(*sensore di presenza alla base dell'ascensore*)
IF NOT (ReadyLoadForVerificationBlockHigh OR ReadyLoadForVerificationBlockLow) AND NOT RotaryMakerInPositionVerificationBlockLow  THEN
	IF LiftPosition<=8 AND ElementVerificationCharged OR (RotaryMakerInPositionVerification AND ElementRotaryCharged)  THEN
			ReadyLoadForVerification:=TRUE;  (*sensore di presenza alla base dell'ascensore*)
		ELSE ReadyLoadForVerification:=FALSE;
	END_IF;
END_IF;
(*caso RotaryMakerInPositionVerificationBlockLow*)
IF NOT (ReadyLoadForVerificationBlockHigh OR ReadyLoadForVerificationBlockLow) AND RotaryMakerInPositionVerificationBlockLow THEN
	IF LiftPosition<=8 AND ElementRotaryCharged AND RotaryPosition=180 THEN
			ReadyLoadForVerification:=TRUE;
	END_IF;
	IF  LiftPosition>8 OR ToExtendCylinderOfExtractionVsGuide THEN
			ReadyLoadForVerification:=FALSE;
	END_IF;
END_IF;

(*sensore di presenza alla base dell'ascensore guasto: *)
IF ReadyLoadForVerificationBlockHigh THEN
	ReadyLoadForVerification:=TRUE;
END_IF;
IF ReadyLoadForVerificationBlockLow THEN
	ReadyLoadForVerification:=FALSE;
END_IF;

(*visualizzazione ElementoMisura*)
IF CylinderUpToMeasureLoad (*.........AND NOT ElementOneTableCharged.........*) AND ElementVerificationCharged AND NOT CylinderUpToMeasureLoadBlockHigh THEN	(*Quando l'ascensore arriva in cima viene reso visibile l'elemento in questa posizione e invisibile quello in posizione di verifica*)
	ElementMeasureCharged:=TRUE;
	ElementMeasureRed:=ElementVerificationRed;
	ElementMeasureSilver:=ElementVerificationSilver;
	ElementMeasureBlack:=ElementVerificationBlack;
	ElementMeasureOverturned:=ElementVerificationOverturned;
	ElementMeasureShort:=ElementVerificationShort;
	ElementVerificationCharged:=FALSE;
END_IF;

(*cuscinetto d'aria*)
IF NOT AirCushionBlock THEN
	IF AirCushion THEN
			 AirCushionVis:=TRUE; (*visualizzazione cuscinetto*)
		ELSE IF NOT AirCushionBlockHigh THEN
				AirCushionVis:=FALSE;
			END_IF;
	END_IF;
END_IF;

(*Elemento cuscinetto d'aria*)
IF (AirCushionVis OR AirCushionBlock) AND (CylinderOfExtractionPosition=80)  THEN	(*Quando e' attiva l'aria dello scivolo e ho spinto il pezzo, viene reso visibile l'elemento in questa posizione e invisibile quello in posizione di misura*)
	ElementAirCharged:=TRUE;
	ElementAirRed:=ElementMeasureRed;
	ElementAirSilver:=ElementMeasureSilver;
	ElementAirBlack:=ElementMeasureBlack;
	ElementAirOverturned:=ElementMeasureOverturned;
	ElementMeasureCharged:=FALSE;
END_IF;

IF (AirCushionVis AND NOT AirCushionBlock) AND (CylinderOfExtractionPosition=80)  AND MovementElementAir<=20  THEN (*Quando l'aria  dello scivolo e' attiva e il pezzo è stato spinto, il pezzo va verso la tavola rotante*)
		MovementElementAir:=MovementElementAir+3;
	ELSE MovementElementAir:=0;
END_IF;

IF (MovementElementAir>=20)
THEN	MovementElementAir:=20;
		ElementAirVsRotaryTable:=TRUE;
		AirCushion:=FALSE;
		ElementAirCharged:=FALSE;
END_IF;

IF NOT Alligneed AND NOT ElementMeasureCharged
THEN	ElementAirRed:=FALSE;
		ElementAirSilver:=FALSE;
		ElementAirBlack:=FALSE;
		ElementMeasureRed:=FALSE;
		ElementMeasureSilver:=FALSE;
		ElementMeasureBlack:=FALSE;
END_IF;

(*---------------------------------------------------------*)
IF (Reset AND NOT MachineNOTOkForReset) OR Remove OR FaultDetected THEN  (*rimozione di tutti i pezzi presenti sulle macchine tramite pulsante o reset del sistema*)
	ElementOneCharged:=FALSE;
	ElementOneRed:=FALSE;
	ElementOneSilver:=FALSE;
	ElementOneBlack:=FALSE;
	ElementOneOverturned:=FALSE;
	ElementOneShort:=FALSE;
	ElementTwoCharged:=FALSE;
	ElementTwoRed:=FALSE;
	ElementTwoSilver:=FALSE;
	ElementTwoBlack:=FALSE;
	ElementTwoOverturned:=FALSE;
	ElementTwoShort:=FALSE;
	ElementThreeCharged:=FALSE;
	ElementThreeRed:=FALSE;
	ElementThreeSilver:=FALSE;
	ElementThreeBlack:=FALSE;
	ElementThreeOverturned:=FALSE;
	ElementThreeShort:=FALSE;
	ElementFourCharged:=FALSE;
	ElementFourRed:=FALSE;
	ElementFourSilver:=FALSE;
	ElementFourBlack:=FALSE;
	ElementFourOverturned:=FALSE;
	ElementFourShort:=FALSE;
	ElementFiveCharged:=FALSE;
	ElementFiveRed:=FALSE;
	ElementFiveSilver:=FALSE;
	ElementFiveBlack:=FALSE;
	ElementFiveOverturned:=FALSE;
	ElementFiveShort:=FALSE;
	ElementSixCharged:=FALSE;
	ElementSixRed:=FALSE;
	ElementSixSilver:=FALSE;
	ElementSixBlack:=FALSE;
	ElementSixOverturned:=FALSE;
	ElementSixShort:=FALSE;
	ElementSevenCharged:=FALSE;
	ElementSevenRed:=FALSE;
	ElementSevenSilver:=FALSE;
	ElementSevenBlack:=FALSE;
	ElementSevenOverturned:=FALSE;
	ElementSevenShort:=FALSE;
	ElementEightCharged:=FALSE;
	ElementEightRed:=FALSE;
	ElementEightSilver:=FALSE;
	ElementEightBlack:=FALSE;
	ElementEightOverturned:=FALSE;
	ElementEightShort:=FALSE;
	ElementWaitingCharged:=FALSE;
	ElementWaitingOverturned:=FALSE;
	ElementWaitingShort:=FALSE;
	ElementRotaryCharged:=FALSE;
	ElementRotaryOverturned:=FALSE;
	ElementRotaryShort:=FALSE;
	ElementVerificationCharged:=FALSE;
	ElementVerificationOverturned:=FALSE;
	ElementVerificationShort:=FALSE;
	ElementMeasureCharged:=FALSE;
	ElementMeasureOverturned:=FALSE;
	ElementMeasureShort:=FALSE;
	ElementAirCharged:=FALSE;
	ElementAirOverturned:=FALSE;
	ElementOneTableCharged:=FALSE;
	ElementOneTableOverturned:=FALSE;

	ElementAirVsRotaryTable:=FALSE;
	ElementAirRed:=FALSE;
	ElementAirBlack:=FALSE;
	ElementAirSilver:=FALSE;
END_IF;
END_PROGRAM

(* POU 0_Simulation/PlantLavorazione, ST *)
PROGRAM PlantLavorazione
VAR

	Set:BOOL:=TRUE;
	FLAG: BOOL := TRUE;
	ElementInControlOverturned: BOOL;
	FLAGRotaryTableMotorBlockHigh: BOOL;
	FLAGToLowerCylinderToInspectLoadBlockHigh: BOOL;
	FLAGBlockingCylinderForwardInDrillingPositioningBlockHigh: BOOL;
	FLAGToLowerDrillingUnitBlockHigh: BOOL;
	FLAGToLiftDrillingUnitBlockHigh: BOOL;
	FLAGExpellingLeverActiveBlockHigh: BOOL;

END_VAR
(*STAZIONE DI LAVORAZIONE - Gestione della Tavola Rotante*)

(*Posizione iniziale della tavola selezionabile mediante pulsante, per simulare una inizializzazione da posizione indefinita*)
IF FLAG
THEN 	FLAG:=FALSE;
		RotaryTableVisual:=RotaryVisIn;	(*variabile di posizione "visuale"*)
		RotaryTablePosition:=RotaryVisIn-30;
END_IF;

(*Attivando il comando di rotazione della tavola rotante, viene incrementata la psozione della tavola *)
IF NOT RotaryTableMotorBlockLow
THEN	IF RotaryTableMotor OR (FLAGRotaryTableMotorBlockHigh AND EmergencyStop)
		THEN	RotaryTablePosition:=RotaryTablePosition+2;
				RotaryTableVisual:=RotaryTableVisual+2;
				IF RotaryTableMotorBlockHigh
				THEN FLAGRotaryTableMotorBlockHigh:=TRUE;
				ELSE FLAGRotaryTableMotorBlockHigh:=FALSE;
				END_IF;

				(*    La posizione viene incrementata ad ogni ciclo del programma, quindi potrebbe verificarsi il superamento della posizione desiderata,
					con le conseguenze di un errato funzionamento del sistema.
                                  A questo proposito ogni volta che viene spento il motore della tavola, vengono settati i corretti valori di posizione*)
		ELSE	IF RotaryTablePosition>357 OR (RotaryTablePosition>-3 AND RotaryTablePosition<3)
				THEN RotaryTablePosition:=0;
						RotaryTableVisual:=30;
				END_IF;
				IF RotaryTablePosition>57 AND RotaryTablePosition<63
				THEN RotaryTablePosition:=60;
						RotaryTableVisual:=90;
				END_IF;
				IF RotaryTablePosition>117 AND RotaryTablePosition<123
				THEN RotaryTablePosition:=120;
						RotaryTableVisual:=150;
				END_IF;
				IF RotaryTablePosition>177 AND RotaryTablePosition<183
				THEN RotaryTablePosition:=180;
						RotaryTableVisual:=210;
				END_IF;
				IF RotaryTablePosition>237 AND RotaryTablePosition<243
				THEN RotaryTablePosition:=240;
						RotaryTableVisual:=270;
				END_IF;
				IF RotaryTablePosition>297 AND RotaryTablePosition<303
				THEN RotaryTablePosition:=300;
						RotaryTableVisual:=330;
				END_IF;
		END_IF;
END_IF;

(*La variabile di spostamento della tavola torna a 0 ogni volta che quest'ultima si muove di 360°*)
IF RotaryTablePosition=360
THEN	RotaryTablePosition:=0;
END_IF;

IF RotaryTableVisual=360
THEN	RotaryTableVisual:=0;
END_IF;
(*Quando una base transita tra stazione di verifica e stazione di lavorazione (passando per la slitta), viene attivata la variabile ElementAirVsRotaryTable.*)
(*Quindi, quando è attiva la variabile ElementAirVsRotaryTable, posso attivare il sensore di presenza che indica l'arrivo di una base nella giostra*)
IF (ElementAirVsRotaryTable AND NOT AvailableLoadForWorkingStationBlockLow) OR AvailableLoadForWorkingStationBlockHigh
THEN	AvailableLoadForWorkingStation:=TRUE;
ELSE   AvailableLoadForWorkingStation:=FALSE;
END_IF;

(*Quando la tavola inizia a muoversi si azzera il sensore di presenza pezzo nella prima stazione*)
IF ((RotaryTablePosition>=1 AND RotaryTablePosition<=2) OR (RotaryTablePosition>=61 AND RotaryTablePosition<=62) OR (RotaryTablePosition>=121 AND RotaryTablePosition<=122) OR (RotaryTablePosition>=181 AND RotaryTablePosition<=182) OR (RotaryTablePosition>=241 AND RotaryTablePosition<=242)) AND NOT AvailableLoadForWorkingStationBlockHigh
THEN   ElementAirVsRotaryTable:=FALSE;
END_IF;

(*Ogni volta che la tavola compie 60°, si attiva il sensore di allineamento della tavola*)
IF AlignementRotaryTableWithPositioningsBlockHigh OR (NOT AlignementRotaryTableWithPositioningsBlockLow AND ((RotaryTablePosition>=-2 AND RotaryTablePosition<=2) OR (RotaryTablePosition>=58 AND RotaryTablePosition<=62) OR (RotaryTablePosition>=118 AND RotaryTablePosition<=122) OR (RotaryTablePosition>=178 AND RotaryTablePosition<=182) OR (RotaryTablePosition>=238 AND RotaryTablePosition<=242) OR (RotaryTablePosition>=298 AND RotaryTablePosition<=302)))
THEN	AlignementRotaryTableWithPositionings:=TRUE;	(*Si attiva il sensore relativo alla posizione della tavola*)
ELSE   AlignementRotaryTableWithPositionings:=FALSE;
END_IF;

(*Utilizzo Alligneed per mettere a true i sensori Available... anche in caso di Fault di AlignementRotary...*)
IF (RotaryTablePosition>=-2 AND RotaryTablePosition<=2) OR (RotaryTablePosition>=58 AND RotaryTablePosition<=62) OR (RotaryTablePosition>=118 AND RotaryTablePosition<=122) OR (RotaryTablePosition>=178 AND RotaryTablePosition<=182) OR (RotaryTablePosition>=238 AND RotaryTablePosition<=242) OR (RotaryTablePosition>=298 AND RotaryTablePosition<=302)
THEN Alligneed:=TRUE;
ELSE Alligneed:=FALSE;
END_IF;

(*Reset dei sensori di controllo e foratura non appena la tavola ha ruotato abbastanza da non essere più allineata*)
IF NOT Alligneed
THEN 	IF NOT AvailableLoadInControlPositioningBlockHigh
		THEN AvailableLoadInControlPositioning:=FALSE;
		END_IF;
		IF NOT AvailableLoadInDrillingPositioningBlockHigh
		THEN AvailableLoadInDrillingPositioning:=FALSE;
		END_IF;
END_IF;


(*********************************************************************************************************************)

(*GESTIONE COLORE DELLE STAZIONI DELLA GIOSTRA*)

(*Reset dei colori dalla posizione di 180°, ovvero dopo l'espulsione dalla giostra*)
(*
ColorCircle[1]=NERO
ColorCircle[2]=BIANCO
ColorCircle[3]=ROSSO
ColorCircle[4]=GRIGIO
*)

IF (ElementSleighCharged OR ExpellingLeverActiveBlockLow OR FLAGExpellingLeverActiveBlockHigh OR AlignementRotaryTableWithPositioningsBlockHigh OR AlignementRotaryTableWithPositioningsBlockLow OR RotaryTableMotorBlockHigh OR Remove)
		(*Non appena viene espulsa la base che era presente nella stazione1 della giostra, ovvero quando la tavola è a 180° e la base è giunta alla slitta tra giostra e robot,
		la circonferenza che rappresenta la stazione1 nella vista dall'alto della tavola, dovrà essere resettata al colore BIANCO*)
THEN 	IF RotaryTablePosition>=180 AND RotaryTablePosition<=200 (*ho messo un range per essere sicuro*)
		THEN Color1:=ColorCircle[2];
				ElementOneTableCharged:=FALSE;
		END_IF;

		(*Non appena viene espulsa la base che era presente nella stazione2 della giostra, ovvero quando la tavola è a 240° e la base è giunta alla slitta tra giostra e robot,
		la circonferenza che rappresenta la stazione2 nella vista dall'alto della tavola, dovrà essere resettata al colore BIANCO*)
		IF RotaryTablePosition>=240 AND RotaryTablePosition<=260
		THEN Color2:=ColorCircle[2];
				ElementTwoTableCharged:=FALSE;
		END_IF;

		IF RotaryTablePosition>=300 AND RotaryTablePosition<=320
		THEN Color3:=ColorCircle[2];
				ElementThreeTableCharged:=FALSE;
		END_IF;

		IF RotaryTablePosition>=0 AND RotaryTablePosition<=20
		THEN Color4:=ColorCircle[2];
				ElementFourTableCharged:=FALSE;
		END_IF;

		IF RotaryTablePosition>=60 AND RotaryTablePosition<=80
		THEN Color5:=ColorCircle[2];
				ElementFiveTableCharged:=FALSE;
		END_IF;

		IF RotaryTablePosition>=120 AND RotaryTablePosition<=140
		THEN Color6:=ColorCircle[2];
				ElementSixTableCharged:=FALSE;
		END_IF;
END_IF;

(*Associo ad ogni stazione un'angolo : stazione1 ==>position=0, stazione2 ==> position=300,
stazione3 ==> position=240, stazione4 ==> position=180, stazione5 ==> position=120 e stazione6 ==> position=60*)

(*Ogni volta ke la tavola è allineata ed è disponibile un pezzo:*)

IF (RotaryTablePosition>=358 OR RotaryTablePosition<=2) AND ElementAirVsRotaryTable (*Quando la stazione1 della tavola è in corrispondenza della slitta tra verifica e lavorazione...*)
THEN	IF ElementAirRed (*Se dalla slitta sta arrivando una base rossa, *)
		THEN Color1:=ColorCircle[3];  (*allora faccio diventare rossa la circonferenza che rappresenta la stazione1 nella giostra vista dall'alto*)
				ElementOneTableRed:=TRUE; (*e attivo la variabile che corrisponde alla presenza di una base rossa nella stazione1 della tavola rotante*)
		ELSE ElementOneTableRed:=FALSE;
		END_IF;
		IF ElementAirSilver (*Se dalla slitta arriva una base argento, *)
		THEN Color1:=ColorCircle[4];  (*allora faccio diventare argento la circonferenza che rappresenta la stazione1 nella giostra vista dall'alto*)
				ElementOneTableSilver:=TRUE;  (*e attivo la variabile che corrisponde alla presenza di una base argento nella stazione1 della tavola rotante*)
		ELSE ElementOneTableSilver:=FALSE;
		END_IF;
		IF ElementAirBlack  (*Se dalla slitta arriva una base nera, *)
		THEN Color1:=ColorCircle[1];    (*allora faccio diventare nera la circonferenza che rappresenta la stazione1 nella giostra vista dall'alto*)
				ElementOneTableBlack:=TRUE;  (*e attivo la variabile che corrisponde alla presenza di una base nera nella stazione1 della tavola rotante*)
		ELSE ElementOneTableBlack:=FALSE;
		END_IF;
		IF ElementAirOverturned  (*Se la base che sta arrivando dalla slitta è Overturned, allora attivo la variabile che corrisponde ad una base Overturned nella stazione1*)
		THEN ElementOneTableOverturned:=TRUE;
		ELSE ElementOneTableOverturned:=FALSE;
		END_IF;
		IF (NOT ElementAirRed AND NOT ElementAirSilver AND NOT ElementAirBlack) (*Se non è in arrivo nessuna base, allora la circonferenza dovrà rimanere bianca*)
		THEN 	Color1:=ColorCircle[2];
				ElementOneTableCharged:=FALSE; (*e la variabile che indica la prsenza di una base nella stazione1 dovrà essere settata a false*)
		ELSE ElementOneTableCharged:=TRUE;
		END_IF;
END_IF;

IF (RotaryTablePosition>=58 AND RotaryTablePosition<=62) AND ElementAirVsRotaryTable
THEN	IF ElementAirRed
		THEN Color2:=ColorCircle[3];
				ElementTwoTableRed:=TRUE;
		ELSE ElementTwoTableRed:=FALSE;
		END_IF;
		IF ElementAirSilver
		THEN Color2:=ColorCircle[4];
				ElementTwoTableSilver:=TRUE;
		ELSE ElementTwoTableSilver:=FALSE;
		END_IF;
		IF ElementAirBlack
		THEN Color2:=ColorCircle[1];
				ElementTwoTableBlack:=TRUE;
		ELSE ElementTwoTableBlack:=FALSE;
		END_IF;
		IF ElementAirOverturned
		THEN ElementTwoTableOverturned:=TRUE;
		ELSE ElementTwoTableOverturned:=FALSE;
		END_IF;
		IF (NOT ElementAirRed AND NOT ElementAirSilver AND NOT ElementAirBlack)
		THEN 	Color2:=ColorCircle[2];
				ElementTwoTableCharged:=FALSE;
		ELSE ElementTwoTableCharged:=TRUE;
		END_IF;
END_IF;

IF (RotaryTablePosition>=118 AND RotaryTablePosition<=122) AND ElementAirVsRotaryTable
THEN	IF ElementAirRed
		THEN Color3:=ColorCircle[3];
				ElementThreeTableRed:=TRUE;
		ELSE ElementThreeTableRed:=FALSE;
		END_IF;
		IF ElementAirSilver
		THEN Color3:=ColorCircle[4];
				ElementThreeTableSilver:=TRUE;
		ELSE ElementThreeTableSilver:=FALSE;
		END_IF;
		IF ElementAirBlack
		THEN Color3:=ColorCircle[1];
				ElementThreeTableBlack:=TRUE;
		ELSE ElementThreeTableBlack:=FALSE;
		END_IF;
		IF ElementAirOverturned
		THEN ElementThreeTableOverturned:=TRUE;
		ELSE ElementThreeTableOverturned:=FALSE;
		END_IF;
		IF (NOT ElementAirRed AND NOT ElementAirSilver AND NOT ElementAirBlack)
		THEN 	Color3:=ColorCircle[2];
				ElementThreeTableCharged:=FALSE;
		ELSE ElementThreeTableCharged:=TRUE;
		END_IF;
END_IF;

IF (RotaryTablePosition>=178 AND RotaryTablePosition<=182) AND ElementAirVsRotaryTable
THEN	IF ElementAirRed
		THEN Color4:=ColorCircle[3];
				ElementFourTableRed:=TRUE;
		ELSE ElementFourTableRed:=FALSE;
		END_IF;
		IF ElementAirSilver
		THEN Color4:=ColorCircle[4];
				ElementFourTableSilver:=TRUE;
		ELSE ElementFourTableSilver:=FALSE;
		END_IF;
		IF ElementAirBlack
		THEN Color4:=ColorCircle[1];
				ElementFourTableBlack:=TRUE;
		ELSE ElementFourTableBlack:=FALSE;
		END_IF;
		IF ElementAirOverturned
		THEN ElementFourTableOverturned:=TRUE;
		ELSE ElementFourTableOverturned:=FALSE;
		END_IF;
		IF (NOT ElementAirRed AND NOT ElementAirSilver AND NOT ElementAirBlack)
		THEN 	Color4:=ColorCircle[2];
				ElementFourTableCharged:=FALSE;
		ELSE ElementFourTableCharged:=TRUE;
		END_IF;
END_IF;

IF (RotaryTablePosition>=238 AND RotaryTablePosition<=242) AND ElementAirVsRotaryTable
THEN	IF ElementAirRed
		THEN Color5:=ColorCircle[3];
				ElementFiveTableRed:=TRUE;
		ELSE ElementFiveTableRed:=FALSE;
		END_IF;
		IF ElementAirSilver
		THEN Color5:=ColorCircle[4];
				ElementFiveTableSilver:=TRUE;
		ELSE ElementFiveTableSilver:=FALSE;
		END_IF;
		IF ElementAirBlack
		THEN Color5:=ColorCircle[1];
				ElementFiveTableBlack:=TRUE;
		ELSE ElementFiveTableBlack:=FALSE;
		END_IF;
		IF ElementAirOverturned
		THEN ElementFiveTableOverturned:=TRUE;
		ELSE ElementFiveTableOverturned:=FALSE;
		END_IF;
		IF (NOT ElementAirRed AND NOT ElementAirSilver AND NOT ElementAirBlack)
		THEN 	Color5:=ColorCircle[2];
				ElementFiveTableCharged:=FALSE;
		ELSE ElementFiveTableCharged:=TRUE;
		END_IF;
END_IF;

IF (RotaryTablePosition>=298 AND RotaryTablePosition<=302) AND ElementAirVsRotaryTable
THEN	IF ElementAirRed
		THEN Color6:=ColorCircle[3];
				ElementSixTableRed:=TRUE;
		ELSE ElementSixTableRed:=FALSE;
		END_IF;
		IF ElementAirSilver
		THEN Color6:=ColorCircle[4];
				ElementSixTableSilver:=TRUE;
		ELSE ElementSixTableSilver:=FALSE;
		END_IF;
		IF ElementAirBlack
		THEN Color6:=ColorCircle[1];
				ElementSixTableBlack:=TRUE;
		ELSE ElementSixTableBlack:=FALSE;
		END_IF;
		IF ElementAirOverturned
		THEN ElementSixTableOverturned:=TRUE;
		ELSE ElementSixTableOverturned:=FALSE;
		END_IF;
		IF (NOT ElementAirRed AND NOT ElementAirSilver AND NOT ElementAirBlack)
		THEN 	Color6:=ColorCircle[2];
				ElementSixTableCharged:=FALSE;
		ELSE ElementSixTableCharged:=TRUE;
		END_IF;
END_IF;

(*Se l'elemento presente nella stazione1 della giostra, è Overturned, allora viene visualizzata la O all'interno della base1*)
IF ElementOneTableOverturned
THEN ElementOneTableO:='O';
ELSE	ElementOneTableO:=' ';
END_IF;

(*Se l'elemento presente nella stazione2 della giostra, è Overturned, allora viene visualizzata la O all'interno della base2*)
IF ElementTwoTableOverturned
THEN ElementTwoTableO:='O';
ELSE	ElementTwoTableO:=' ';
END_IF;

IF ElementThreeTableOverturned
THEN ElementThreeTableO:='O';
ELSE	ElementThreeTableO:=' ';
END_IF;

IF ElementFourTableOverturned
THEN ElementFourTableO:='O';
ELSE	ElementFourTableO:=' ';
END_IF;

IF ElementFiveTableOverturned
THEN ElementFiveTableO:='O';
ELSE	ElementFiveTableO:=' ';
END_IF;

IF ElementSixTableOverturned
THEN ElementSixTableO:='O';
ELSE	ElementSixTableO:=' ';
END_IF;

(*********************************************************************************************************************)


(*Simulazione del funzionamento del sensore di presenza nella stazione di foratura*)
IF RotaryTablePosition=60
THEN IF  (ElementOneTableCharged AND NOT AvailableLoadInControlPositioningBlockLow) OR AvailableLoadInControlPositioningBlockHigh
		THEN 	AvailableLoadInControlPositioning:=TRUE;
				IF InspectPosition=InspectDepth AND ((NOT ElementOneTableOverturned AND NOT InControlLoadInWrongPositionToBeDrilledBlockLow) OR InControlLoadInWrongPositionToBeDrilledBlockHigh)
				THEN 	InControlLoadInWrongPositionToBeDrilled:=TRUE;
				ELSE 	InControlLoadInWrongPositionToBeDrilled:=FALSE;
				END_IF;
		ELSE 	IF NOT AvailableLoadInControlPositioningBlockHigh
				THEN AvailableLoadInControlPositioning:=FALSE;
				END_IF;
		END_IF;
END_IF;

IF RotaryTablePosition=120
THEN IF  (ElementTwoTableCharged AND NOT AvailableLoadInControlPositioningBlockLow) OR AvailableLoadInControlPositioningBlockHigh
		THEN 	AvailableLoadInControlPositioning:=TRUE;
				IF InspectPosition=InspectDepth AND ((NOT ElementTwoTableOverturned AND NOT InControlLoadInWrongPositionToBeDrilledBlockLow) OR InControlLoadInWrongPositionToBeDrilledBlockHigh)
				THEN 	InControlLoadInWrongPositionToBeDrilled:=TRUE;
				ELSE 	InControlLoadInWrongPositionToBeDrilled:=FALSE;
				END_IF;
		ELSE	IF NOT AvailableLoadInControlPositioningBlockHigh
				THEN AvailableLoadInControlPositioning:=FALSE;
				END_IF;
		END_IF;
END_IF;

IF RotaryTablePosition=180
THEN IF  (ElementThreeTableCharged AND NOT AvailableLoadInControlPositioningBlockLow) OR AvailableLoadInControlPositioningBlockHigh
		THEN 	AvailableLoadInControlPositioning:=TRUE;
				IF InspectPosition=InspectDepth AND ((NOT ElementThreeTableOverturned AND NOT InControlLoadInWrongPositionToBeDrilledBlockLow) OR InControlLoadInWrongPositionToBeDrilledBlockHigh)
				THEN 	InControlLoadInWrongPositionToBeDrilled:=TRUE;
				ELSE 	InControlLoadInWrongPositionToBeDrilled:=FALSE;
				END_IF;
		ELSE   IF NOT AvailableLoadInControlPositioningBlockHigh
				THEN AvailableLoadInControlPositioning:=FALSE;
				END_IF;
		END_IF;
END_IF;

IF RotaryTablePosition=240
THEN IF  (ElementFourTableCharged AND NOT AvailableLoadInControlPositioningBlockLow) OR AvailableLoadInControlPositioningBlockHigh
		THEN 	AvailableLoadInControlPositioning:=TRUE;
				IF InspectPosition=InspectDepth AND ((NOT ElementFourTableOverturned AND NOT InControlLoadInWrongPositionToBeDrilledBlockLow) OR InControlLoadInWrongPositionToBeDrilledBlockHigh)
				THEN	InControlLoadInWrongPositionToBeDrilled:=TRUE;
				ELSE	InControlLoadInWrongPositionToBeDrilled:=FALSE;
				END_IF;
		ELSE 	IF NOT AvailableLoadInControlPositioningBlockHigh
				THEN AvailableLoadInControlPositioning:=FALSE;
				END_IF;
		END_IF;
END_IF;

IF RotaryTablePosition=300
THEN IF  (ElementFiveTableCharged AND NOT AvailableLoadInControlPositioningBlockLow) OR AvailableLoadInControlPositioningBlockHigh
		THEN 	AvailableLoadInControlPositioning:=TRUE;
				IF InspectPosition=InspectDepth AND ((NOT ElementFiveTableOverturned AND NOT InControlLoadInWrongPositionToBeDrilledBlockLow) OR InControlLoadInWrongPositionToBeDrilledBlockHigh)
				THEN 	InControlLoadInWrongPositionToBeDrilled:=TRUE;
				ELSE 	InControlLoadInWrongPositionToBeDrilled:=FALSE;
				END_IF;
		ELSE 	IF NOT AvailableLoadInControlPositioningBlockHigh
				THEN AvailableLoadInControlPositioning:=FALSE;
				END_IF;
		END_IF;
END_IF;

IF RotaryTablePosition=0
THEN IF (ElementSixTableCharged AND NOT AvailableLoadInControlPositioningBlockLow) OR AvailableLoadInControlPositioningBlockHigh
		THEN 	AvailableLoadInControlPositioning:=TRUE;
				IF InspectPosition=InspectDepth AND ((NOT ElementSixTableOverturned AND NOT InControlLoadInWrongPositionToBeDrilledBlockLow) OR InControlLoadInWrongPositionToBeDrilledBlockHigh)
				THEN 	InControlLoadInWrongPositionToBeDrilled:=TRUE;
				ELSE 	InControlLoadInWrongPositionToBeDrilled:=FALSE;
				END_IF;
		ELSE 	IF NOT AvailableLoadInControlPositioningBlockHigh
				THEN AvailableLoadInControlPositioning:=FALSE;
				END_IF;
		END_IF;
END_IF;

(*Bloccaggio alto indipendente dalla posizione della tavola*)
IF FLAGInControlLoadInWrongPositionToBeDrilled (*settaggio del FLAG a righa 485 *)
THEN InControlLoadInWrongPositionToBeDrilled:=TRUE;
END_IF;

IF AvailableLoadInControlPositioningBlockHigh
THEN AvailableLoadInControlPositioning:=TRUE;
END_IF;

IF AvailableLoadInControlPositioningBlockLow
THEN AvailableLoadInControlPositioning:=FALSE;
END_IF;

(*FORATURA*)
(*---------------------------------------------------------------------------------------------------------------------------*)

(*Quando la tavola raggiunge i 120°, se è presente un pezzo nella stazione1, si attiva il sensore di presenza presente nella stazione di foratura *)
IF RotaryTablePosition=120
THEN IF (ElementOneTableCharged AND NOT AvailableLoadInDrillingPositioningBlockLow) OR AvailableLoadInDrillingPositioningBlockHigh
		THEN 	AvailableLoadInDrillingPositioning:=TRUE;
		ELSE 	IF NOT AvailableLoadInDrillingPositioningBlockHigh
				THEN AvailableLoadInDrillingPositioning:=FALSE;
				END_IF;
		END_IF;
END_IF;
(*Quando la tavola raggiunge i 180°, se è presente un pezzo nella stazione2, si attiva il sensore di presenza presente nella stazione di foratura *)
IF RotaryTablePosition=180
THEN IF (ElementTwoTableCharged AND NOT AvailableLoadInDrillingPositioningBlockLow) OR AvailableLoadInDrillingPositioningBlockHigh
		THEN 	AvailableLoadInDrillingPositioning:=TRUE;
		ELSE	IF NOT AvailableLoadInDrillingPositioningBlockHigh
				THEN AvailableLoadInDrillingPositioning:=FALSE;
				END_IF;
		END_IF;
END_IF;

IF RotaryTablePosition=240
THEN IF  (ElementThreeTableCharged AND NOT AvailableLoadInDrillingPositioningBlockLow) OR AvailableLoadInDrillingPositioningBlockHigh
		THEN 	AvailableLoadInDrillingPositioning:=TRUE;
		ELSE 	IF NOT AvailableLoadInDrillingPositioningBlockHigh
				THEN AvailableLoadInDrillingPositioning:=FALSE;
				END_IF;
		END_IF;
END_IF;

IF RotaryTablePosition=300
THEN IF  (ElementFourTableCharged AND NOT AvailableLoadInDrillingPositioningBlockLow) OR AvailableLoadInDrillingPositioningBlockHigh
		THEN 	AvailableLoadInDrillingPositioning:=TRUE;
		ELSE	IF NOT AvailableLoadInDrillingPositioningBlockHigh
				THEN AvailableLoadInDrillingPositioning:=FALSE;
				END_IF;
		END_IF;
END_IF;

IF RotaryTablePosition=0
THEN IF  (ElementFiveTableCharged AND NOT AvailableLoadInDrillingPositioningBlockLow) OR AvailableLoadInDrillingPositioningBlockHigh
		THEN 	AvailableLoadInDrillingPositioning:=TRUE;
		ELSE 	IF NOT AvailableLoadInDrillingPositioningBlockHigh
				THEN AvailableLoadInDrillingPositioning:=FALSE;
				END_IF;
		END_IF;
END_IF;

IF RotaryTablePosition=60
THEN IF (ElementSixTableCharged AND NOT AvailableLoadInDrillingPositioningBlockLow) OR AvailableLoadInDrillingPositioningBlockHigh
		THEN 	AvailableLoadInDrillingPositioning:=TRUE;
		ELSE 	IF NOT AvailableLoadInDrillingPositioningBlockHigh
				THEN AvailableLoadInDrillingPositioning:=FALSE;
				END_IF;
		END_IF;
END_IF;

IF  AvailableLoadInDrillingPositioningBlockHigh
THEN  AvailableLoadInDrillingPositioning:=TRUE;
END_IF;

IF  AvailableLoadInDrillingPositioningBlockLow
THEN  AvailableLoadInDrillingPositioning:=FALSE;
END_IF;

(*--------------------------------------------------------------------------------------------------------------------------------*)


(*STAZIONE DI CONTROLLO*)
(*------------------------------------------------------------------------------------------------------*)
(*Se l'elemento che si trova nella stazione di controllo è Overturned, allora la variabile ElementInControlOverturned:=TRUE*)
IF (RotaryTablePosition =60 AND ElementOneTableOverturned) OR (RotaryTablePosition =120 AND ElementTwoTableOverturned) OR (RotaryTablePosition =180 AND ElementThreeTableOverturned) OR (RotaryTablePosition =240 AND ElementFourTableOverturned) OR (RotaryTablePosition =300 AND ElementFiveTableOverturned) OR (RotaryTablePosition =0 AND ElementSixTableOverturned) AND NOT InControlLoadInWrongPositionToBeDrilledBlockHigh
THEN ElementInControlOverturned:=TRUE;
ELSE ElementInControlOverturned:=FALSE;
END_IF;
(*Se la base è Overturned, allora la profondità a cui andrà l'utensile di controllo è minore rispetto al caso di una base corretta*)
IF ElementInControlOverturned
THEN InspectDepth:=9;
ELSE InspectDepth:=18;
END_IF;

(*Simulazione del tastatore*)
(*Se viene dato il comando di abbassare la torretta di controllo, allora la variabile associata alla posizione della torretta, viene incrementata, altrimenti essa viene decrementata*)
IF FLAGToLowerCylinderToInspectLoadBlockHigh OR (ToLowerCylinderToInspectLoad AND NOT ToLowerCylinderToInspectLoadBlockLow)
THEN InspectPosition:=InspectPosition+2;
		IF ToLowerCylinderToInspectLoadBlockHigh
		THEN FLAGToLowerCylinderToInspectLoadBlockHigh:=TRUE;
		ELSE FLAGToLowerCylinderToInspectLoadBlockHigh:=FALSE;
		END_IF;
ELSE  InspectPosition:=InspectPosition-2;
END_IF;

(*Quando l'utensile raggiunge la profondità desiderata, si impone il non superamento di essa*)
IF InspectPosition>=InspectDepth
THEN	InspectPosition:=InspectDepth;
END_IF;

IF InspectPosition<=0
THEN InspectPosition:=0;
END_IF;
(*---------------------------------------------------------------------------------------*)


(*FORATURA*)
(*-----------------------------------------------------------------------------*)
(*Se il trapano è attivo, allora l'utensile in visualizzazione cambia colore*)
IF DrillingUnitActiveBlockHigh OR (DrillingUnitActive AND NOT DrillingUnitActiveBlockLow)
THEN DrillingToolColor:=TRUE;
ELSE DrillingToolColor:=FALSE;
END_IF;

(*Se viene attivato il pistone di bloccaggio del pezzo, nella stazione di foratura, allora viene incrementata la posizione di esso, finchè non raggiunge il fine corsa superiore*)
IF FLAGBlockingCylinderForwardInDrillingPositioningBlockHigh OR (BlockingCylinderForwardInDrillingPositioning AND NOT BlockingCylinderForwardInDrillingPositioningBlockLow)
THEN 	IF BlockingActuator<24
		THEN BlockingActuator:=BlockingActuator+7;
		ELSE BlockingActuator:=24;
		END_IF;
		IF BlockingCylinderForwardInDrillingPositioningBlockHigh
		THEN FLAGBlockingCylinderForwardInDrillingPositioningBlockHigh:=TRUE;
		ELSE FLAGBlockingCylinderForwardInDrillingPositioningBlockHigh:=FALSE;
		END_IF;
(*Decemento della posizione del pistone, sino all'arrivo al fine corsa inferiore*)
ELSE 	IF BlockingActuator>0
		THEN BlockingActuator:=BlockingActuator-7;
		ELSE BlockingActuator:=0;
		END_IF;
END_IF;

(*Simulazione operazione di foratura*)

(*Se viene richiesto di abbassare la torretta di foratura, allora la variabile associata alla posizione della torretta viene incrementata*)
IF FLAGToLowerDrillingUnitBlockHigh OR (ToLowerDrillingUnit AND NOT ToLowerDrillingUnitBlockLow)
THEN DrillingUnitPosition:=DrillingUnitPosition+2;
		IF ToLowerDrillingUnitBlockHigh
		THEN FLAGToLowerDrillingUnitBlockHigh:=TRUE;
		ELSE FLAGToLowerDrillingUnitBlockHigh:=FALSE;
		END_IF;
END_IF;
(*Se viene richiesto di sollevare la torretta di foratura, allora la variabile di posizione viene decrementata*)
IF FLAGToLiftDrillingUnitBlockHigh OR (ToLiftDrillingUnit AND NOT ToLiftDrillingUnitBlockLow)
THEN DrillingUnitPosition:=DrillingUnitPosition-2;
		IF ToLiftDrillingUnitBlockHigh
		THEN FLAGToLiftDrillingUnitBlockHigh:=TRUE;
		ELSE FLAGToLiftDrillingUnitBlockHigh:=FALSE;
		END_IF;
END_IF;

(*Quando la torretta giunge al fine corsa inferiore, si attiva il sensore di presenza inferiore "DrillingUnitDown" *)
IF DrillingUnitPosition>=22
THEN 	DrillingUnitPosition:=22;
END_IF;

IF ToLowerDrillingUnit
THEN 	IF DrillingUnitPosition>=20
		THEN 	IF NOT DrillingUnitDownBlockLow
				THEN	DrillingUnitDown:=TRUE;
				ELSE 	DrillingUnitDown:=FALSE;
				END_IF;
		END_IF;
ELSE 	IF NOT DrillingUnitDownBlockHigh
		THEN DrillingUnitDown:=FALSE;
		END_IF;
END_IF;

(*Quando la torretta raggiunge il fine corsa superiore, si attiva il sensore di presenza superiore "DrillingUnitUp" *)
IF DrillingUnitPosition<=0
THEN 	DrillingUnitPosition:=0;
END_IF;

IF ToLiftDrillingUnit
THEN	IF DrillingUnitPosition<3
		THEN	IF NOT DrillingUnitUpBlockLow
				THEN DrillingUnitUp:=TRUE;
				ELSE DrillingUnitUp:=FALSE;
				END_IF;
		END_IF;
ELSE 	IF NOT DrillingUnitUpBlockHigh
		THEN DrillingUnitUp:=FALSE;
		END_IF;
END_IF;

IF DrillingUnitUpBlockHigh
THEN  DrillingUnitUp:=TRUE;
END_IF;
IF DrillingUnitDownBlockHigh
THEN  DrillingUnitDown:=TRUE;
END_IF;
IF DrillingUnitUpBlockHigh
THEN  DrillingUnitUp:=TRUE;
END_IF;
IF DrillingUnitDownBlockLow
THEN  DrillingUnitDown:=FALSE;
END_IF;

(*------------------------------------------------------------------------------------*)


(*INCREMENTO DELLE VARIABILI ASSOCIATE ALLA POSIZIONE LINEARE DELLE BASI SULLA GIOSTRA*)

IF RotaryTablePosition>0 AND RotaryTablePosition<=180 (*Tra 0-180° la base deve traslare orizzontalmente dalla posizione iniziale a quella di espulsione*)
THEN 	LinearTablePosition1:=RotaryTablePosition*1.4; (*LinearTablePosition1 è la variabile di posizione associata alla base1, ed è proporzionale alla posizione della tavola rotante, con un fattore di 1,4. Quest'ultimo è stato ricavato imponendo che la base raggiunga la posizione di espulsione al raggiungimento dei 180° *)
ELSE LinearTablePosition1:=0; (*Quando la base viene espulsa, essa diventa invisibile e quindi può essere riportata alla posizione iniziale*)
END_IF;

IF RotaryTablePosition>60 AND RotaryTablePosition<=240
THEN 	LinearTablePosition2:=(RotaryTablePosition-60)*1.4;
ELSE LinearTablePosition2:=0;
END_IF;

IF RotaryTablePosition>120 AND RotaryTablePosition<=300
THEN 	LinearTablePosition3:=(RotaryTablePosition-120)*1.4;
ELSE LinearTablePosition3:=0;
END_IF;

(*CASI PARTICOLARI DOVUTI AL FATTO CHE QUANDO RotaryTable=360 ==> RotaryTable:=0*)
(*--------------------------------------------------------------------------------------------------------------------------------------*)
IF RotaryTablePosition>180 AND (RotaryTablePosition<=360 OR RotaryTablePosition=0)
THEN 	LinearTablePosition4:=ABS(RotaryTablePosition-180)*1.4; (*ABS è il valore assoluto. Esso è necessario dal momento in cui RotaryTablePosition=0,  per ottenere una posizione lineare positiva*)
END_IF;

IF RotaryTablePosition>2 AND RotaryTablePosition<=180
THEN LinearTablePosition4:=0;
END_IF;

IF RotaryTablePosition>240 AND (RotaryTablePosition<=360 OR RotaryTablePosition=0)
THEN LinearTablePosition5:=ABS(RotaryTablePosition-240)*1.4;
END_IF;

IF (RotaryTablePosition>2 AND RotaryTablePosition<=60)
THEN LinearTablePosition5:=(RotaryTablePosition+120)*1.4;
END_IF;

IF (RotaryTablePosition>60 AND RotaryTablePosition<=240)
THEN LinearTablePosition5:=0;
END_IF;

IF RotaryTablePosition>300 AND (RotaryTablePosition<=360 OR RotaryTablePosition=0)
THEN LinearTablePosition6:=ABS(RotaryTablePosition-300)*1.4;
END_IF;

IF (RotaryTablePosition>2 AND RotaryTablePosition<=120)
THEN LinearTablePosition6:=(RotaryTablePosition+60)*1.4;
END_IF;

IF (RotaryTablePosition>120 AND RotaryTablePosition<=300)
THEN LinearTablePosition6:=0;
END_IF;
(*---------------------------------------------------------------------------------------------------------------------------------------*)

(*Stazione di Espulsione*)

(*Buffer per riportare l'informazione alla slitta prima del robot*)
IF RotaryTablePosition=180 (*Quando la tavola è a 180°, allora viene espulsa la base1*)
THEN 	ElementSleighRed:=ElementOneTableRed; (*BUFFER che trasferisce le informazioni della base che si trova nella stazione di espulsione, alla slitta tra giostra e robot *)
		ElementSleighBlack:=ElementOneTableBlack;
		ElementSleighSilver:=ElementOneTableSilver;
		ElementSleighOverturned:=ElementOneTableOverturned;
		IF ElementOneTableCharged (*Se è presente una base nella stazione di espulsione, allora viene attivato il sensore "virtuale" di presenza*)
		THEN 	AvailableLoadInExpulsionPositioning:=TRUE; (*Sensore "virtuale, perchè non prensente veramente nell'impianto" settato a true*)
		END_IF;
END_IF;

IF RotaryTablePosition=240 (*Quando la tavola è a 240°, allora viene espulsa la base2*)
THEN 	ElementSleighRed:=ElementTwoTableRed;
		ElementSleighBlack:=ElementTwoTableBlack;
		ElementSleighSilver:=ElementTwoTableSilver;
		ElementSleighOverturned:=ElementTwoTableOverturned;
		IF ElementTwoTableCharged
		THEN 	AvailableLoadInExpulsionPositioning:=TRUE;
		END_IF;
END_IF;

IF RotaryTablePosition=300
THEN 	ElementSleighRed:=ElementThreeTableRed;
		ElementSleighBlack:=ElementThreeTableBlack;
		ElementSleighSilver:=ElementThreeTableSilver;
		ElementSleighOverturned:=ElementThreeTableOverturned;
		IF ElementThreeTableCharged
		THEN 	AvailableLoadInExpulsionPositioning:=TRUE;
		END_IF;
END_IF;

IF RotaryTablePosition=0
THEN 	ElementSleighRed:=ElementFourTableRed;
		ElementSleighBlack:=ElementFourTableBlack;
		ElementSleighSilver:=ElementFourTableSilver;
		ElementSleighOverturned:=ElementFourTableOverturned;
		IF ElementFourTableCharged
		THEN 	AvailableLoadInExpulsionPositioning:=TRUE;
		END_IF;
END_IF;

IF RotaryTablePosition=60
THEN 	ElementSleighRed:=ElementFiveTableRed;
		ElementSleighBlack:=ElementFiveTableBlack;
		ElementSleighSilver:=ElementFiveTableSilver;
		ElementSleighOverturned:=ElementFiveTableOverturned;
		IF ElementFiveTableCharged
		THEN 	AvailableLoadInExpulsionPositioning:=TRUE;
		END_IF;
END_IF;

IF RotaryTablePosition=120
THEN 	ElementSleighRed:=ElementSixTableRed;
		ElementSleighBlack:=ElementSixTableBlack;
		ElementSleighSilver:=ElementSixTableSilver;
		ElementSleighOverturned:=ElementSixTableOverturned;
		IF ElementSixTableCharged
		THEN 	AvailableLoadInExpulsionPositioning:=TRUE;
		END_IF;
END_IF;

(*Se l'elemento presente nella slitta di espulsione tra giostra e robot, è Overturned, allora viene visualizzata la O all'interno della base*)
IF ElementSleighOverturned
THEN ElementSleighO:='O';
ELSE	ElementSleighO:=' ';
END_IF;

(*Attivando la leva di espulsione, viene incrementata la sua posizione*)
IF FLAGExpellingLeverActiveBlockHigh OR (ExpellingLeverActive AND NOT ExpellingLeverActiveBlockLow)
THEN	LeverPosition:=LeverPosition+10;
		IF ExpellingLeverActiveBlockHigh
		THEN FLAGExpellingLeverActiveBlockHigh:=TRUE;
		ELSE FLAGExpellingLeverActiveBlockHigh:=FALSE;
		END_IF;
ELSE	LeverPosition:=LeverPosition-10;
END_IF;

IF LeverPosition<0
THEN	LeverPosition:=0;
END_IF;

(*Se il cilindro di espulsione raggiunge il fine corsa, il pezzo e' pronto per l'assemblaggio*)
IF LeverPosition>=50
THEN	LeverPosition:=50;
		ElementSleighCharged:=TRUE;
END_IF;

(*Quando è presente un pezzo sulla slitta, viene incrementata la sua posizione*)
IF ElementSleighCharged
THEN MovementElementSleigh:=MovementElementSleigh+2;
ELSE MovementElementSleigh:=0;
END_IF;

(*Quando la base raggiunge la fine della slitta, viene resa invisibile, passando le sue informazioni e rendendo visibile la base nella "Stazione1" (da qui indicherò con Stazione1 la stazione dopo la giostra)*)
IF (MovementElementSleigh>=10)
THEN	MovementElementSleigh:=10;
		ElementSleighCharged:=FALSE;
		ElementStation1RobotCharged:=TRUE;
		ElementStation1RobotRed:=ElementSleighRed;
		ElementStation1RobotBlack:=ElementSleighBlack;
		ElementStation1RobotSilver:=ElementSleighSilver;
		ElementStation1RobotOverturned:=ElementSleighOverturned;
		IF NOT AvailableLoadForRobotBlockLow
		THEN AvailableLoadForRobot:=TRUE; (*si attiva il sensore di presenza pezzo nella stazione tra giostra e robot*)
		END_IF;
END_IF;

IF AvailableLoadForRobotBlockHigh
THEN AvailableLoadForRobot:=TRUE;
END_IF;

(*Se la base presente nella Stazione1 è Overturned, rendo visibile la O all'interno di essa.*)
IF ElementStation1RobotOverturned
THEN ElementStation1RobotO:='O';
ELSE ElementStation1RobotO:='';
END_IF;


IF Remove
THEN	Color1:=ColorCircle[2];
		Color2:=ColorCircle[2];
		Color3:=ColorCircle[2];
		Color4:=ColorCircle[2];
		Color5:=ColorCircle[2];
		Color6:=ColorCircle[2];
		ElementAirVsRotaryTable:=FALSE;
		ElementMeasureCharged:=FALSE;
		AlignementRotaryTableWithPositionings:=FALSE;
		AvailableLoadForWorkingStation:=FALSE;
		AvailableLoadInControlPositioning:=FALSE;
		AvailableLoadInDrillingPositioning:=FALSE;
		AvailableLoadInExpulsionPositioning:=FALSE;
		InControlLoadInWrongPositionToBeDrilled:=FALSE;
		LeverPosition:=0;
		ElementSleighRed:=FALSE;
		ElementSleighBlack:=FALSE;
		ElementSleighSilver:=FALSE;
		ElementSleighCharged:=FALSE;
		ElementSleighOverturned:=FALSE;
		ElementOneTableCharged:=FALSE;
		ElementTwoTableCharged:=FALSE;
		ElementThreeTableCharged:=FALSE;
		ElementFourTableCharged:=FALSE;
		ElementFiveTableCharged:=FALSE;
		ElementSixTableCharged:=FALSE;
END_IF;

IF FaultDetected
THEN 	FLAGRotaryTableMotorBlockHigh:=FALSE;
		FLAGToLowerCylinderToInspectLoadBlockHigh:=FALSE;
		FLAGBlockingCylinderForwardInDrillingPositioningBlockHigh:=FALSE;
		FLAGToLowerDrillingUnitBlockHigh:=FALSE;
		FLAGToLiftDrillingUnitBlockHigh:=FALSE;
		FLAGExpellingLeverActiveBlockHigh:=FALSE;
END_IF;
END_PROGRAM

(* POU 0_Simulation/PlantAssemblaggio, ST *)
PROGRAM PlantAssemblaggio
VAR
	State: INT;
	Count: BOOL;
	Count2: BOOL;
	CaseBlack: INT;
	CaseRedSilver: INT;
	CaseOverturned: INT;
	InitialPosition: INT;
	FLAGToExtractSpringInAssemblyStationBlockHigh: BOOL;
	FLAGBlockingCylinderForwardInAssemblyStationBlockHigh: BOOL;
	FLAGToExtractCoverInAssemblyStationForwardBlockHigh: BOOL;
	Count3: BOOL;
	Count4: BOOL;
END_VAR
(*QUANDO UN PEZZO E' STATO ASSEMBLATO, RESETTO TUTTI I CONTATORI*)
IF ElementAssembled
THEN	CanDiscard:=FALSE; (*RENDE INVISIBILE IL CESTO PORTA SCARTI*)
		ElementToDiscard:=FALSE; (*RESET DELLE PROPRIETA' DEL PEZZO NEL CESTO DEGLI SCARTI*)
		ElementToDiscardRed:=FALSE;
		ElementToDiscardBlack:=FALSE;
		ElementToDiscardSilver:=FALSE;
		ElementToDiscardPosition:=0;
		CoverToDiscard:=FALSE;
		PistonBlackToDiscard:=FALSE;
		PistonSilverToDiscard:=FALSE;
		ElementAssembled:=FALSE;
END_IF;

(*Premendo il tasto FillWarehouse, si simula il riempimento di tutti i magazzini*)
IF FillAllWarehouses
THEN 	SpringLoad:=TRUE;
		CoverLoad:=TRUE;
		PistonLoad:=TRUE;
		FillAllWarehouses:=FALSE;
END_IF;


(*MODULO MOLLE*)

(*Tasto che serve a caricare le molle nel magazzino*)
IF SpringLoad
THEN	SpringNumber:=8;
		Spring1:=TRUE;
		Spring2:=TRUE;
		Spring3:=TRUE;
		Spring4:=TRUE;
		Spring5:=TRUE;
		Spring6:=TRUE;
		Spring7:=TRUE;
		Spring8:=TRUE;
		SpringLoad:=FALSE;
END_IF;

(*NB: IL CILINDRO DI ESTRAZIONE E' NORMALMENTE APERTO!!!*)
(*Quando il comando di estrazione è TRUE, lo stelo del cilindro rientra*)
IF FLAGToExtractSpringInAssemblyStationBlockHigh OR (ToExtractSpringInAssemblyStation AND NOT ToExtractSpringInAssemblyStationBlockLow)
THEN	ExtractSpringPosition:=ExtractSpringPosition-4;
		IF ToExtractSpringInAssemblyStationBlockHigh
		THEN FLAGToExtractSpringInAssemblyStationBlockHigh:=TRUE;
		ELSE FLAGToExtractSpringInAssemblyStationBlockHigh:=FALSE;
		END_IF;
ELSE	ExtractSpringPosition:=ExtractSpringPosition+4;
END_IF;

(*Quando il pistone di estrazione molle e' arrivato a fine corsa, viene resa visibile la molla estratta*)
IF ExtractSpringPosition<=0
THEN	ExtractSpringPosition:=0;

		IF NOT ToExtractSpringInAssemblyStationInRetroactivePositionBlockLow
		THEN ToExtractSpringInAssemblyStationInRetroactivePosition:=TRUE;
		ELSE ToExtractSpringInAssemblyStationInRetroactivePosition:=FALSE;
		END_IF;

		IF SpringNumber>0 (*se il magazzino molle non è vuoto*)
		THEN VisualSpring:=TRUE; (*allora rendo visibile la molla che trasla insieme al pistone di prelievo molle*)
		END_IF;

ELSE	IF NOT ToExtractSpringInAssemblyStationInRetroactivePositionBlockHigh
		THEN ToExtractSpringInAssemblyStationInRetroactivePosition:=FALSE;
		ELSE ToExtractSpringInAssemblyStationInRetroactivePosition:=TRUE;
		END_IF;

IF ToExtractSpringInAssemblyStationInRetroactivePositionBlockHigh
THEN ToExtractSpringInAssemblyStationInRetroactivePosition:=TRUE;
END_IF;

END_IF;

(*Quando il pistone di estrazione molle e' in posizione di riposo, si attiva il relativo sensore e si disattiva il flag "SpringBehind", che indica il movimento verso il riposo del pistone*)
IF ExtractSpringPosition>=40
THEN	ExtractSpringPosition:=40;

		IF NOT ToExtractSpringInAssemblyStationInExtensivePositionBlockLow
		THEN ToExtractSpringInAssemblyStationInExtensivePosition:=TRUE;
		ELSE ToExtractSpringInAssemblyStationInExtensivePosition:=FALSE;
		END_IF;

		VisualSpring:=FALSE;
		IF Count
		THEN 	SpringNumber:=SpringNumber-1;
				SpringExtract:=TRUE;
				Count:=FALSE;
		END_IF;

ELSE	IF NOT ToExtractSpringInAssemblyStationInExtensivePositionBlockHigh
		THEN ToExtractSpringInAssemblyStationInExtensivePosition:=FALSE;
		ELSE ToExtractSpringInAssemblyStationInExtensivePosition:=TRUE;
		END_IF;
		Count:=TRUE;
END_IF;

IF ToExtractSpringInAssemblyStationInExtensivePositionBlockHigh
THEN ToExtractSpringInAssemblyStationInExtensivePosition:=TRUE;
END_IF;

IF SpringNumber=7 (*AND ToExtractSpringInAssemblyStationInRetroactivePosition*)
THEN Spring8:=FALSE;
END_IF;
IF SpringNumber=6
THEN Spring7:=FALSE;
END_IF;
IF SpringNumber=5
THEN Spring6:=FALSE;
END_IF;
IF SpringNumber=4
THEN Spring5:=FALSE;
END_IF;
IF SpringNumber=3
THEN Spring4:=FALSE;
END_IF;
IF SpringNumber=2
THEN Spring3:=FALSE;
END_IF;
IF SpringNumber=1
THEN Spring2:=FALSE;
END_IF;
IF SpringNumber=0
THEN 	Spring1:=FALSE;
END_IF;


(*MODULO PISTONI*)

IF PistonLoad
THEN 	PistonBlackLoad:=TRUE;
		PistonSilverLoad:=TRUE;
		PistonLoad:=FALSE;
END_IF;

(*Quando attiviamo questa variabile, riempiamo il magazzino pistoni neri*)
IF PistonBlackLoad
THEN	PistonBlackNumber:=8;
		PistonBlack1:=TRUE;
		PistonBlack2:=TRUE;
		PistonBlack3:=TRUE;
		PistonBlack4:=TRUE;
		PistonBlack5:=TRUE;
		PistonBlack6:=TRUE;
		PistonBlack7:=TRUE;
		PistonBlack8:=TRUE;
		PistonBlackLoad:=FALSE;
END_IF;

(*Quando attiviamo questa variabile, riempiamo il magazzino pistoni grigi*)
IF PistonSilverLoad
THEN	PistonSilverNumber:=8;
		PistonSilver1:=TRUE;
		PistonSilver2:=TRUE;
		PistonSilver3:=TRUE;
		PistonSilver4:=TRUE;
		PistonSilver5:=TRUE;
		PistonSilver6:=TRUE;
		PistonSilver7:=TRUE;
		PistonSilver8:=TRUE;
		PistonSilverLoad:=FALSE;
END_IF;

(*DA COMMENTARE...*)
	IF PistonSelectorIsOnTheRight
	THEN	PistonBlack8:=FALSE;
	END_IF;

	IF PistonSelectorIsOnTheLeft
	THEN	PistonSilver8:=FALSE;
	END_IF;

(*La sottrazione del pistone viene fatta dall'end-effector*)
IF PistonSelectorPosition=20
THEN	IF PistonSilverNumber=7
		THEN	PistonSilver7:=FALSE;
		END_IF;

		IF PistonSilverNumber=6
		THEN	PistonSilver6:=FALSE;
		END_IF;

		IF PistonSilverNumber=5
		THEN	PistonSilver5:=FALSE;
		END_IF;

		IF PistonSilverNumber=4
		THEN	PistonSilver4:=FALSE;
		END_IF;

		IF PistonSilverNumber=3
		THEN	PistonSilver3:=FALSE;
		END_IF;

		IF PistonSilverNumber=2
		THEN	PistonSilver2:=FALSE;
		END_IF;

		IF PistonSilverNumber=1
		THEN	PistonSilver1:=FALSE;
		END_IF;
END_IF;

IF PistonSelectorPosition=-20
THEN	IF PistonBlackNumber=7
		THEN	PistonBlack7:=FALSE;
		END_IF;

		IF PistonBlackNumber=6
		THEN	PistonBlack6:=FALSE;
		END_IF;

		IF PistonBlackNumber=5
		THEN	PistonBlack5:=FALSE;
		END_IF;

		IF PistonBlackNumber=4
		THEN	PistonBlack4:=FALSE;
		END_IF;

		IF PistonBlackNumber=3
		THEN	PistonBlack3:=FALSE;
		END_IF;

		IF PistonBlackNumber=2
		THEN	PistonBlack2:=FALSE;
		END_IF;

		IF PistonBlackNumber=1
		THEN	PistonBlack1:=FALSE;
		END_IF;
END_IF;

(*Incremento di posizione verso sinistra*)
IF PistonSelectorGoOnTheLeftBlockHigh OR (PistonSelectorGoOnTheLeft AND NOT PistonSelectorGoOnTheLeftBlockLow)
THEN	PistonSelectorPosition:=PistonSelectorPosition+3;
END_IF;
(*Incremento di posizione verso destra*)
IF PistonSelectorGoOnTheRightBlockHigh OR (PistonSelectorGoOnTheRight AND NOT PistonSelectorGoOnTheRightBlockLow)
THEN	PistonSelectorPosition:=PistonSelectorPosition-3;
END_IF;

(*Quando l'incremento di posizione giunge a 20 siamo in corrsipondenza del fine corsa destro*)
IF PistonSelectorPosition<=-20
THEN PistonSelectorPosition:=-20;
		(*Se il sensore di posizione destro non è bloccato alto, allora il sensore è attivo*)
		IF NOT PistonSelectorIsOnTheRightBlockLow
		THEN PistonSelectorIsOnTheRight:=TRUE;
		ELSE PistonSelectorIsOnTheRight:=FALSE;
		END_IF;
		(*Se il magazzino pistoni grigi non è vuoto, allora visualizzo il  pistone all'interno del selettore*)
		IF PistonBlackNumber>0
		THEN PistonBlackExtract:=TRUE;
		END_IF;

ELSE 	IF NOT PistonSelectorIsOnTheRightBlockHigh
		THEN PistonSelectorIsOnTheRight:=FALSE;
		END_IF;
END_IF;

IF PistonSelectorIsOnTheRightBlockHigh
THEN PistonSelectorIsOnTheRight:=TRUE;
END_IF;

IF PistonSelectorPosition>=20
THEN PistonSelectorPosition:=20;

		IF NOT PistonSelectorIsOnTheLeftBlockLow
		THEN PistonSelectorIsOnTheLeft:=TRUE;
		ELSE PistonSelectorIsOnTheLeft:=FALSE;
		END_IF;

		IF PistonSilverNumber>0
		THEN PistonSilverExtract:=TRUE;
		END_IF;

ELSE	IF NOT PistonSelectorIsOnTheLeftBlockHigh
		THEN PistonSelectorIsOnTheLeft:=FALSE;
		END_IF;
END_IF;

IF PistonSelectorIsOnTheLeftBlockHigh
THEN PistonSelectorIsOnTheLeft:=TRUE;
END_IF;


(*MODULO COPERCHI*)

IF CoverLoad
THEN	CoverNumber:=8;
		IF NOT EmptyCoverHouseInAssemblyStationBlockHigh
		THEN EmptyCoverHouseInAssemblyStation:=FALSE;
		END_IF;
		Cover1:=TRUE;
		Cover2:=TRUE;
		Cover3:=TRUE;
		Cover4:=TRUE;
		Cover5:=TRUE;
		Cover6:=TRUE;
		Cover7:=TRUE;
		Cover8:=TRUE;
		CoverLoad:=FALSE;
END_IF;

IF FLAGToExtractCoverInAssemblyStationForwardBlockHigh OR (ToExtractCoverInAssemblyStationForward AND NOT ToExtractCoverInAssemblyStationForwardBlockLow)
THEN	ExtractCoverPosition:=ExtractCoverPosition+3;
		IF ToExtractCoverInAssemblyStationForwardBlockHigh
		THEN FLAGToExtractCoverInAssemblyStationForwardBlockHigh:=TRUE;
		ELSE FLAGToExtractCoverInAssemblyStationForwardBlockHigh:=FALSE;
		END_IF;
ELSE	ExtractCoverPosition:=ExtractCoverPosition-3;
END_IF;

IF ExtractCoverPosition<=0
THEN	ExtractCoverPosition:=0;
		IF NOT ToExtractCoverInAssemblyStationInRetroactivePositionBlockLow
		THEN ToExtractCoverInAssemblyStationInRetroactivePosition:=TRUE;
		ELSE ToExtractCoverInAssemblyStationInRetroactivePosition:=FALSE;
		END_IF;

		IF NOT EmptyCoverHouseInAssemblyStation
		THEN Cover1:=TRUE;
		END_IF;

ELSE	IF NOT ToExtractCoverInAssemblyStationInRetroactivePositionBlockHigh
		THEN ToExtractCoverInAssemblyStationInRetroactivePosition:=FALSE;
		ELSE ToExtractCoverInAssemblyStationInRetroactivePosition:=TRUE;
		END_IF;
END_IF;

IF ExtractCoverPosition>=65
THEN	ExtractCoverPosition:=65;
		Cover1:=FALSE;
		IF Count2
		THEN 	CoverNumber:=CoverNumber-1;
				CoverExtract:=TRUE;
				Count2:=FALSE;
		END_IF;

		IF NOT ToExtractCoverInAssemblyStationInExtensivePositionBlockLow
		THEN ToExtractCoverInAssemblyStationInExtensivePosition:=TRUE;
		ELSE ToExtractCoverInAssemblyStationInExtensivePosition:=FALSE;
		END_IF;

ELSE	IF NOT ToExtractCoverInAssemblyStationInExtensivePositionBlockHigh
		THEN ToExtractCoverInAssemblyStationInExtensivePosition:=FALSE;
		ELSE ToExtractCoverInAssemblyStationInExtensivePosition:=TRUE;
		END_IF;
		Count2:=TRUE;
END_IF;

IF  ToExtractCoverInAssemblyStationInRetroactivePositionBlockHigh
THEN ToExtractCoverInAssemblyStationInRetroactivePosition:=TRUE;
END_IF;

IF ToExtractCoverInAssemblyStationInExtensivePositionBlockHigh
THEN ToExtractCoverInAssemblyStationInExtensivePosition:=TRUE;
END_IF;


IF ExtractCoverPosition=0
THEN	IF CoverNumber=7
		THEN	Cover8:=FALSE;
		END_IF;
		IF CoverNumber=6
		THEN	Cover7:=FALSE;
		END_IF;
		IF CoverNumber=5
		THEN	Cover6:=FALSE;
		END_IF;
		IF CoverNumber=4
		THEN	Cover5:=FALSE;
		END_IF;
		IF CoverNumber=3
		THEN	Cover4:=FALSE;
		END_IF;
		IF CoverNumber=2
		THEN	Cover3:=FALSE;
		END_IF;
		IF CoverNumber=1
		THEN	Cover2:=FALSE;
		END_IF;
		IF CoverNumber=0
		THEN	Cover1:=FALSE;
				IF NOT EmptyCoverHouseInAssemblyStationBlockLow
				THEN EmptyCoverHouseInAssemblyStation:=TRUE;
				ELSE EmptyCoverHouseInAssemblyStation:=FALSE;
				END_IF;
		END_IF;
END_IF;

IF EmptyCoverHouseInAssemblyStationBlockHigh
THEN EmptyCoverHouseInAssemblyStation:=TRUE;
END_IF;


(*SIMULAZIONE DEI MOVIMENTI DEL ROBOT *)
(*________________________________________________________________________________________________________*)
(*
(*Bloccaggio basso degli attuatori "robot"*)
IF RobotTakeLoadToDiascardBlockLow OR RobotTakeRedSilverLoadBlockLow OR RobotTakeBlackLoadBlockLow OR RobotGoToInitialPositionBlockLow OR RobotGoToSpringHouseBlockLow OR RobotGoToPistonHouseBlockLow OR RobotGoToCoverHouseBlockLow OR RobotTakeCurrentLoadToAssemblyBlockLow
THEN RobotBitIn3:=FALSE; RobotBitIn2:=FALSE; RobotBitIn1:=FALSE; RobotBitIn0:=FALSE;
END_IF;
*)
IF Bit4Output
THEN State:=0;
END_IF;

(*Spingendo il tasto StopProgramRunning, simulo lo spegnimento del programma CosiRop*)
IF StopProgramRunning
THEN RobotProgramRunning:=FALSE;
ELSE RobotProgramRunning:=TRUE;
END_IF;


IF RobotProgramRunning
THEN
		(*Se si riceve il comando di prelievo di una base capovolta(Base Nera 0101, Base Rossa-Argento 0100) *)
		IF RobotTakeLoadToDiascardBlockHigh OR ((NOT Bit3Output AND Bit2Output AND NOT Bit1Output) AND NOT RobotTakeLoadToDiascardBlockLow)
		THEN	State:=1;
		END_IF;

		(*Se si riceve il comando di prelievo di una Base Nera 0010 *)
		IF RobotTakeBlackLoadBlockHigh OR ((NOT Bit3Output AND NOT Bit2Output AND Bit1Output  AND NOT Bit0Output) AND NOT RobotTakeBlackLoadBlockLow)
		THEN	State:=2;
		END_IF;

		(*Se si riceve il comando di prelievo di una Base Rossa-Argento 0011 *)
		IF RobotTakeRedSilverLoadBlockHigh OR ((NOT Bit3Output AND NOT Bit2Output AND Bit1Output AND Bit0Output) AND NOT RobotTakeRedSilverLoadBlockLow)
		THEN	State:=3;
		END_IF;

		IF (NOT Bit3Output AND NOT Bit2Output AND NOT Bit1Output AND Bit0Output) AND State=0
		THEN State:=4;
		END_IF;
END_IF;


CASE State OF
(*Lo stato "0" rappresenta lo stato di Idle*)
0:	CaseOverturned:=20;
	CaseBlack:=20;
	CaseRedSilver:=20;
	InitialPosition:=20;

(*Lo stato "1" rappresenta il caso di comando di prelievo di una base Overturned*)
1:	CASE CaseOverturned OF
								(*Da posizione iniziale a stazione1 per prelevare la base*)
						20:		IF NOT RobotEngineBlockLow (*Se non ci sono guasti nei motori del robot, allora il robot comincia a muoversi*)
								THEN RobotGoVerticalPosition:=RobotGoVerticalPosition+10; (*SCENDI SECONDO LA DIREZIONE VERTICALE*)
								END_IF;
								IF NOT RobotInInitialPositionBlockHigh (*Se non c'è un bloccaggio alto del sensoe virtuale di posizione iniziale, allora...*)
								THEN Bit3Input:=FALSE; Bit2Input:=FALSE; Bit1Input:=FALSE; Bit0Input:=FALSE; (*RobotInInitialPosition:=FALSE*)
								END_IF;
								IF RobotGoVerticalPosition>=170
								THEN	RobotGoVerticalPosition:=170;
										CaseOverturned:=21;
								END_IF;
								(*Presa della base*)
						21:		EndEffectorPosition:=EndEffectorPosition+1; (*CHIUDI END-EFFECTOR*)
								IF EndEffectorPosition>=3
								THEN 	EndEffectorPosition:=3;
										CaseOverturned:=22;
								END_IF;
								(*Buffer di trasferimento delle informazioni relative alla base*)
						22:		ElementInEndEffector:=TRUE; (*MOSTRA LA BASE NELL'END-EFFECTOR*)
								ElementInEndEffectorBlack:=ElementStation1RobotBlack;
								ElementInEndEffectorSilver:=ElementStation1RobotSilver;
								ElementInEndEffectorRed:=ElementStation1RobotRed;
								ElementInEndEffectorOverturned:=ElementStation1RobotOverturned;
								IF ElementInEndEffectorOverturned
								THEN ElementInEndEffectorO:='O';
								ELSE ElementInEndEffectorO:='';
								END_IF;
								CaseOverturned:=23;

						23:		ElementStation1RobotCharged:=FALSE;
								CaseOverturned:=24;

						24:		IF NOT RobotEngineBlockLow
								THEN RobotGoVerticalPosition:=RobotGoVerticalPosition-10; (*SALI SECONDO LA DIREZIONE VERTICALE*)
								END_IF;
								IF RobotGoVerticalPosition<=0
								THEN	RobotGoVerticalPosition:=0;
										CaseOverturned:=25;
								END_IF;
								(*RESETTO LE INFORMAZIONI ALLA STAZIONE1 PRIMA DI METTERE A FALSE AvailableLoadForRobot IN MODO DA AVERE LE GIUSTE INFORMAZIONI SUL PEZZO SUCCESSIVO*)
						25:		ElementStation1RobotRed:=FALSE;
								ElementStation1RobotBlack:=FALSE;
								ElementStation1RobotSilver:=FALSE;
								ElementStation1RobotOverturned:=FALSE;
								IF NOT AvailableLoadForRobotBlockHigh
								THEN	AvailableLoadForRobot:=FALSE; (*RESET DEL SENSORE DI PRESENZA NELLA STAZIONE1, A QUESTO PUNTO LA GIOSTRA PUO' MANDARE UN'ALTRO PEZZO*)
								END_IF;
								CaseOverturned:=26;

						26:		CanText:='Scarti'; (*Mostra il testo "scarti" all'interno del cesto*)
								CanColour:=FALSE; (*Quando CanColour è FALSE, il colore del cesto è rosso. Quando è TRUE il colore del cesto è verde*)
								CanDiscard:=TRUE; (*VARIABILE DI VISUALIZZAZIONE: rende visibile il cesto contenente gli scarti*)
								CaseOverturned:=27;
								(*Ritorno alla posizione iniziale*)
						27:		IF NOT RobotEngineBlockLow
								THEN RobotGoHorizontalPosition:=RobotGoHorizontalPosition+10; (*MUOVITI ORIZZONTALMENTE VERSO DESTRA*)
								END_IF;
								IF RobotGoHorizontalPosition>=100
								THEN 	RobotGoHorizontalPosition:=100;
										CaseOverturned:=28;
								END_IF;
								(*MOSTRA IL PEZZO CHE FINIRA' NELLA STAZIONE DI SCARTO*)
						28:		ElementToDiscard:=TRUE;
								IF ElementInEndEffectorOverturned
								THEN ElementToDiscardO:='O';
								END_IF;
								ElementToDiscardRed:=ElementInEndEffectorRed;
								ElementToDiscardBlack:=ElementInEndEffectorBlack;
								ElementToDiscardSilver:=ElementInEndEffectorSilver;
								CaseOverturned:=29;


						29:		EndEffectorPosition:=EndEffectorPosition-1; (*APRI END-EFFECTOR*)
								IF EndEffectorPosition<=0
								THEN 	EndEffectorPosition:=0;
										CaseOverturned:=30;
								END_IF;
								(*RESET DELLE BASI NELL'END-EFFECTOR, NON L'HO FATTO NELL'IF PRECEDENTE PERCHE' AVREI RESO INVISIBILI LE BASI NELLA STAZIONE SCARTI*)
						30:		ElementInEndEffector:=FALSE; (*RENDO INVISIBILE LA BASE NELL'END-EFFECTOR*)
								ElementInEndEffectorRed:=FALSE;
								ElementInEndEffectorBlack:=FALSE;
								ElementInEndEffectorSilver:=FALSE;
								ElementInEndEffectorOverturned:=FALSE;
								CaseOverturned:=31;

						31:		ElementToDiscardPosition:=ElementToDiscardPosition+5; (*lo scarto scende fino a finire nel cestino*)
								IF ElementToDiscardPosition>=80
								THEN 	ElementToDiscardPosition:=80;
										CaseOverturned:=32;
								END_IF;

						32:		IF NOT RobotEngineBlockLow
								THEN RobotGoHorizontalPosition:=RobotGoHorizontalPosition-5; (*MUOVITI ORIZZONTALMENTE VERSO SINISTRA*)
								END_IF;
								IF RobotGoHorizontalPosition<=0
								THEN 	RobotGoHorizontalPosition:=0;
										CaseOverturned:=33;
								END_IF;

						33:		ElementAssembled:=TRUE;
								IF NOT RobotInInitialPositionBlockLow
								THEN Bit1Input:=TRUE; Bit0Input:=TRUE; (*RobotInInitialPosition:=TRUE;*)
								END_IF;
								State:=0;

	END_CASE;



2:	CASE CaseBlack OF

							(*Preleva la base nera*)
						20:		IF NOT RobotEngineBlockLow
								THEN RobotGoVerticalPosition:=RobotGoVerticalPosition+10; (*SCENDI SECONDO LA DIREZIONE VERTICALE*)
								END_IF;
								IF RobotGoVerticalPosition>=170
								THEN	RobotGoVerticalPosition:=170;
										CaseBlack:=21;
								END_IF;

						21:		EndEffectorPosition:=EndEffectorPosition+1; (*CHIUDI END-EFFECTOR*)
								IF EndEffectorPosition>=3
								THEN 	EndEffectorPosition:=3;
										CaseBlack:=22;
								END_IF;

						22:		ElementInEndEffector:=TRUE; (*MOSTRA LA BASE NELL'END-EFFECTOR*)
								ElementInEndEffectorBlack:=ElementStation1RobotBlack;
								ElementInEndEffectorSilver:=ElementStation1RobotSilver;
								ElementInEndEffectorRed:=ElementStation1RobotRed;
								ElementInEndEffectorOverturned:=ElementStation1RobotOverturned;
								IF ElementInEndEffectorOverturned
								THEN ElementInEndEffectorO:='O';
								ELSE ElementInEndEffectorO:='';
								END_IF;
								CaseBlack:=23;

						23:		ElementStation1RobotCharged:=FALSE;
								CaseBlack:=24;

						24:		IF NOT RobotEngineBlockLow
								THEN RobotGoVerticalPosition:=RobotGoVerticalPosition-10; (*SALI SECONDO LA DIREZIONE VERTICALE*)
								END_IF;
								IF RobotGoVerticalPosition<=0
								THEN	RobotGoVerticalPosition:=0;
										CaseBlack:=25;
								END_IF;
								(*RESETTO LE INFORMAZIONI ALLA STAZIONE1 PRIMA DI METTERE A FALSE AvailableLoadForRobot IN MODO DA AVERE LE GIUSTE INFORMAZIONI SUL PEZZO SUCCESSIVO*)
						25:		ElementStation1RobotRed:=FALSE;
								ElementStation1RobotBlack:=FALSE;
								ElementStation1RobotSilver:=FALSE;
								ElementStation1RobotOverturned:=FALSE;
								IF NOT AvailableLoadForRobotBlockHigh
								THEN AvailableLoadForRobot:=FALSE; (*RESET DEL SENSORE DI PRESENZA NELLA STAZIONE1, A QUESTO PUNTO LA GIOSTRA PUO' MANDARE UN'ALTRO PEZZO*)
								END_IF;
								CaseBlack:=26;

						26 :	IF NOT RobotEngineBlockLow
								THEN RobotGoHorizontalPosition:=RobotGoHorizontalPosition+10; (*MUOVITI ORIZZONTALMENTE VERSO DESTRA*)
								END_IF;
								IF RobotGoHorizontalPosition>=100
								THEN	RobotGoHorizontalPosition:=100;
										CaseBlack:=27;
								END_IF;

						27 :	IF NOT RobotEngineBlockLow
								THEN RobotGoVerticalPosition:=RobotGoVerticalPosition+10; (*SCENDI SECONDO LA DIREZIONE VERTICALE*)
								END_IF;
								IF RobotGoVerticalPosition>=190
								THEN 	RobotGoVerticalPosition:=190;
										CaseBlack:=28;
								END_IF;

						28 :	EndEffectorPosition:=EndEffectorPosition-1; (*APRI END-EFFECTOR*)
								IF EndEffectorPosition<=0
								THEN	EndEffectorPosition:=0;
										CaseBlack:=29;
								END_IF;

						29:		ElementAssemblyCharged:=TRUE; (*MOSTRA LA BASE NELLA STAZIONE DI ASSEMBLAGGIO*)
								ElementAssemblyBlack:=ElementInEndEffectorBlack;
								ElementAssemblySilver:=ElementInEndEffectorSilver;
								ElementAssemblyRed:=ElementInEndEffectorRed;
								CaseBlack:=30;


						30 :	ElementInEndEffector:=FALSE; (*NASCONDI LA BASE SULL'END-EFFECTOR*)
								ElementInEndEffectorBlack:=FALSE;
								ElementInEndEffectorSilver:=FALSE;
								ElementInEndEffectorRed:=FALSE;
								ElementInEndEffectorOverturned:=FALSE;
								IF NOT RobotInAssemblyUnitBlockLow AND NOT RobotInInitialPositionBlockHigh
								THEN Bit3Input:=TRUE; Bit2Input:=FALSE; Bit1Input:=FALSE; Bit0Input:=FALSE; (*1000 = RobotInAssemblyUnit*)
								END_IF;
								CaseBlack:=31;

						31:		IF (NOT Bit3Output AND Bit2Output AND Bit1Output AND Bit0Output) AND NOT RobotGoToPistonHouseBlockLow  (*0111 = Prendi Pistone*)
								THEN CaseBlack:=32;
								ELSE CaseBlack:=31;
								END_IF;

						32 :	IF NOT RobotEngineBlockLow
								THEN RobotGoVerticalPosition:=RobotGoVerticalPosition-10;
								END_IF;
								IF NOT RobotInAssemblyUnitBlockHigh
								THEN Bit3Input:=FALSE; (*RobotInAssemblyUnit:=FALSE*)
								END_IF;
								IF RobotGoVerticalPosition<=-90
								THEN	RobotGoVerticalPosition:=-90;
										CaseBlack:=33;
								END_IF;

							(*CHIUDI END-EFFECTOR PER POTER PASSARE TRA LE DUE TORRETTE DEI PISTONI*)
						33 :	EndEffectorPosition:=EndEffectorPosition+1;
								IF EndEffectorPosition>=20
								THEN 	EndEffectorPosition:=20;
										CaseBlack:=34;
								END_IF;

						34 :	IF NOT RobotEngineBlockLow
								THEN RobotGoHorizontalPosition:=RobotGoHorizontalPosition+10;
								END_IF;
								IF RobotGoHorizontalPosition>=280
								THEN 	RobotGoHorizontalPosition:=280;
										CaseBlack:=35;
								END_IF;

						35 : 	IF NOT RobotEngineBlockLow
								THEN RobotGoVerticalPosition:=RobotGoVerticalPosition+10;
								END_IF;
								IF RobotGoVerticalPosition>=230
								THEN	RobotGoVerticalPosition:=230;
										CaseBlack:=36;
								END_IF;

							(*CHIUDI END-EFFECTOR PER PRESA PISTONE*)
						36 :	EndEffectorPosition:=EndEffectorPosition+2;
								IF EndEffectorPosition>=25
								THEN 	EndEffectorPosition:=25;
										CaseBlack:=37;
								END_IF;

						37:		IF PistonSilverExtract AND PistonSelectorPosition=-20(*NOT PistonSelectorIsOnTheRightBlockHigh AND NOT PistonSelectorIsOnTheRightBlockLow AND NOT PistonSelectorIsOnTheLeftBlockHigh AND NOT PistonSelectorIsOnTheLeftBlockLow AND NOT PistonSelectorGoOnTheRightBlockHigh AND NOT PistonSelectorGoOnTheRightBlockLow AND NOT PistonSelectorGoOnTheLeftBlockHigh AND NOT PistonSelectorGoOnTheLeftBlockLow*)
								THEN	PistonSilverInEndEffector:=TRUE; (*RENDO VISIBILE IL PISTONE GRIGIO NELL'END-EFFECTOR*)
										PistonSilverExtract:=FALSE; (*RENDO INVISIBILE IL PISTONE GRIGIO NEL MAGAZZINO*)
										PistonSilverNumber:=PistonSilverNumber-1;
								END_IF;
								IF NOT RobotInPistonWarehouseBlockLow
								THEN Bit0Input:=TRUE; (*RobotInPistonWarehouse:=TRUE;*)
								END_IF;
								CaseBlack:=38;

						38:		IF (Bit3Output AND NOT Bit2Output AND NOT Bit1Output AND Bit0Output) AND NOT RobotTakeCurrentLoadToAssemblyBlockLow   (*1001 = TakeCurrentLoadToAssemblyStation*)
								THEN CaseBlack:=39;
								ELSE CaseBlack:=38;
								END_IF;

						39 :	IF NOT RobotEngineBlockLow
								THEN RobotGoVerticalPosition:=RobotGoVerticalPosition-10;
								END_IF;
								IF NOT RobotInPistonWarehouseBlockHigh
								THEN Bit0Input:=FALSE; (*RobotInPistonWarehouse:=FALSE;*)
								END_IF;
								IF RobotGoVerticalPosition<=-90
								THEN	RobotGoVerticalPosition:=-90;
										CaseBlack:=40;
								END_IF;

						40 :	IF NOT RobotEngineBlockLow
								THEN RobotGoHorizontalPosition:=RobotGoHorizontalPosition-10;
								END_IF;
								IF RobotGoHorizontalPosition<=100
								THEN 	RobotGoHorizontalPosition:=100;
										CaseBlack:=41;
								END_IF;

						41 :	IF NOT RobotEngineBlockLow
								THEN RobotGoVerticalPosition:=RobotGoVerticalPosition+10;
								END_IF;
								IF RobotGoVerticalPosition>=185
								THEN	RobotGoVerticalPosition:=185;
										CaseBlack:=42;
								END_IF;

						42 :	EndEffectorPosition:=EndEffectorPosition-2; (*APRO END-EFFECTOR*)
								IF EndEffectorPosition<=16
								THEN 	EndEffectorPosition:=16;
										PistonBlackAssembly:=PistonBlackInEndEffector;
										PistonSilverAssembly:=PistonSilverInEndEffector;
										CaseBlack:=43;
								END_IF;

						43 :	PistonBlackInEndEffector:=FALSE;
								PistonSilverInEndEffector:=FALSE;
								IF NOT RobotInAssemblyUnitBlockLow
								THEN Bit3Input:=TRUE;  (*RobotInAssemblyUnit:=TRUE;*)
								END_IF;
								CaseBlack:=44;

						44:		IF (NOT Bit3Output AND Bit2Output AND Bit1Output  AND NOT Bit0Output) AND NOT RobotGoToSpringHouseBlockLow   (*0110 = RobotGoToSpringHouse*)
								THEN CaseBlack:=45;
								ELSE CaseBlack:=44;
								END_IF;

						45 :	IF NOT RobotEngineBlockLow
								THEN RobotGoVerticalPosition:=RobotGoVerticalPosition-10;
								END_IF;
								IF NOT RobotInAssemblyUnitBlockHigh
								THEN Bit3Input:=FALSE; (*RobotInAssemblyUnit:=FALSE*)
								END_IF;
								IF RobotGoVerticalPosition<=170
								THEN	RobotGoVerticalPosition:=170;
										CaseBlack:=46;
								END_IF;

						46 :	IF NOT RobotEngineBlockLow
								THEN RobotGoHorizontalPosition:=RobotGoHorizontalPosition+10;
								END_IF;
								IF RobotGoHorizontalPosition>=170
								THEN 	RobotGoHorizontalPosition:=170;
										CaseBlack:=47;
								END_IF;

						47 : 	IF NOT RobotEngineBlockLow
								THEN RobotGoVerticalPosition:=RobotGoVerticalPosition+10;
								END_IF;
								IF RobotGoVerticalPosition>=245
								THEN	RobotGoVerticalPosition:=245;
										CaseBlack:=48;
								END_IF;

						48 :	EndEffectorPosition:=EndEffectorPosition+2; (*CHIUDI END-EFFECTOR PER PRESA MOLLA*)
								IF EndEffectorPosition>=20
								THEN 	EndEffectorPosition:=20;
										CaseBlack:=49;
								END_IF;

						49:		IF NOT ToExtractSpringInAssemblyStationInExtensivePositionBlockHigh AND NOT ToExtractSpringInAssemblyStationInExtensivePositionBlockLow AND NOT ToExtractSpringInAssemblyStationBlockLow AND NOT ToExtractSpringInAssemblyStationBlockHigh
								THEN 	SpringInEndEffector:=TRUE; (*RENDO VISIBILE LA MOLLA NELL'END-EFFECTOR*)
										SpringExtract:=FALSE; (*RENDO INVISIBILE LA MOLLA NEL MAGAZZINO*)
								END_IF;
								IF NOT RobotInSpringWarehouseBlockLow
								THEN Bit1Input:=TRUE; (*RobotInSpringWarehouse:=TRUE;*)
								END_IF;
								CaseBlack:=50;

						50:		IF (Bit3Output AND NOT Bit2Output AND NOT Bit1Output AND Bit0Output) AND NOT RobotTakeCurrentLoadToAssemblyBlockLow  (*1001 = TakeCurrentLoadToAssemblyStation*)
								THEN CaseBlack:=51;
								ELSE CaseBlack:=50;
								END_IF;

						51 :	IF NOT RobotEngineBlockLow
								THEN RobotGoVerticalPosition:=RobotGoVerticalPosition-10;
								END_IF;
								IF NOT RobotInSpringWarehouseBlockHigh
								THEN Bit1Input:=FALSE; (*RobotInSpringWarehouse:=FALSE;*)
								END_IF;
								IF RobotGoVerticalPosition<=140
								THEN	RobotGoVerticalPosition:=140;
										CaseBlack:=52;
								END_IF;

						52 :	IF NOT RobotEngineBlockLow
								THEN RobotGoHorizontalPosition:=RobotGoHorizontalPosition-10;
								END_IF;
								IF RobotGoHorizontalPosition<=100
								THEN 	RobotGoHorizontalPosition:=100;
										CaseBlack:=53;
								END_IF;

						53 : 	IF NOT RobotEngineBlockLow
								THEN RobotGoVerticalPosition:=RobotGoVerticalPosition+10;
								END_IF;
								IF RobotGoVerticalPosition>=180
								THEN	RobotGoVerticalPosition:=180;
										CaseBlack:=54;
								END_IF;

						54 :	EndEffectorPosition:=EndEffectorPosition-2; (*APERTURA END-EFFECTOR*)
								IF EndEffectorPosition<=16
								THEN 	EndEffectorPosition:=16;
										CaseBlack:=55;
								END_IF;

						55:		IF NOT ToExtractSpringInAssemblyStationInExtensivePositionBlockHigh AND NOT ToExtractSpringInAssemblyStationInExtensivePositionBlockLow AND NOT ToExtractSpringInAssemblyStationBlockLow AND NOT ToExtractSpringInAssemblyStationBlockHigh
								THEN 	SpringInEndEffector:=FALSE; (*RENDO INVISIBILE LA MOLLA NELL'END-EFFECTOR*)
										SpringAssembly:=TRUE; (*RENDO VISIBILE LA MOLLA DENTRO LA BASE NELLA STAZIONE DI ASSEMBLAGGIO*)
								END_IF;
								IF NOT RobotInAssemblyUnitBlockLow
								THEN Bit3Input:=TRUE; (*1000 = RobotInAssemblyUnit*)
								END_IF;
								CaseBlack:=56;

						56:		IF (Bit3Output AND NOT Bit2Output AND NOT Bit1Output AND NOT Bit0Output) AND NOT RobotGoToCoverHouseBlockLow  (*1000 = RobotGoToCoverHouse*)
								THEN CaseBlack:=57;
								ELSE CaseBlack:=56;
								END_IF;

						57 :	IF NOT RobotEngineBlockLow
								THEN RobotGoVerticalPosition:=RobotGoVerticalPosition-10;
								END_IF;
								IF NOT RobotInAssemblyUnitBlockHigh
								THEN Bit3Input:=FALSE; (*RobotInAssemblyUnit:=FALSE;*)
								END_IF;
								IF RobotGoVerticalPosition<=-110
								THEN	RobotGoVerticalPosition:=-110;
										CaseBlack:=58;
								END_IF;

						58 :	EndEffectorPosition:=EndEffectorPosition-2; (*APERTURA END-EFFECTOR*)
								IF EndEffectorPosition<=0
								THEN 	EndEffectorPosition:=0;
										CaseBlack:=59;
								END_IF;

						59 :	IF NOT RobotEngineBlockLow
								THEN RobotGoHorizontalPosition:=RobotGoHorizontalPosition+10;
								END_IF;
								IF RobotGoHorizontalPosition>=500
								THEN 	RobotGoHorizontalPosition:=500;
										CaseBlack:=60;
								END_IF;

						60 : 	IF NOT RobotEngineBlockLow
								THEN RobotGoVerticalPosition:=RobotGoVerticalPosition+10;
								END_IF;
								IF RobotGoVerticalPosition>=250
								THEN	RobotGoVerticalPosition:=250;
										CaseBlack:=61;
								END_IF;

						61 :	EndEffectorPosition:=EndEffectorPosition+1; (*CHIUDI END-EFFECTOR PER PRESA MOLLA*)
								IF EndEffectorPosition>=3
								THEN 	EndEffectorPosition:=3;
										CaseBlack:=62;
								END_IF;

						62:		IF NOT ToExtractCoverInAssemblyStationForwardBlockLow AND NOT Count3
								THEN 	CoverInEndEffector:=TRUE; (*RENDO VISIBILE IL COPERCHIO NEL END-EFFECTOR*)
										CoverExtract:=FALSE; (*RENDO INVISIBILE IL COPERCHIO NEL MAGAZZINO*)
										IF ToExtractCoverInAssemblyStationForwardBlockHigh OR ToExtractCoverInAssemblyStationInExtensivePositionBlockHigh
										THEN Count3:=TRUE; (*Count3 è un contatore, necessario per far sì che in caso di bloccaggio alto venga visualizzato il primo coperchio estratto e non i successivi*)
										END_IF;
								END_IF;
								IF NOT RobotInCoverWarehouseBlockLow
								THEN Bit2Input:=TRUE; (*RobotInCoverWarehouse:=TRUE;*)
								END_IF;
								CaseBlack:=63;

						63:		IF (Bit3Output AND NOT Bit2Output AND NOT Bit1Output AND Bit0Output) AND NOT RobotTakeCurrentLoadToAssemblyBlockLow   (*1001 = TakeCurrentLoadToAssemblyStation*)
								THEN CaseBlack:=64;
								ELSE CaseBlack:=63;
								END_IF;

						64 :	IF NOT RobotEngineBlockLow
								THEN RobotGoVerticalPosition:=RobotGoVerticalPosition-10;
								END_IF;
								IF NOT RobotInCoverWarehouseBlockHigh
								THEN Bit2Input:=FALSE; (*RobotInCoverWarehouse:=FALSE;*)
								END_IF;
								IF RobotGoVerticalPosition<=-110
								THEN	RobotGoVerticalPosition:=-110;
										CaseBlack:=65;
								END_IF;

						65 :	IF NOT RobotEngineBlockLow
								THEN RobotGoHorizontalPosition:=RobotGoHorizontalPosition-10;
								END_IF;
								IF RobotGoHorizontalPosition<=100
								THEN 	RobotGoHorizontalPosition:=100;
										CaseBlack:=66;
								END_IF;

						66 : 	IF NOT RobotEngineBlockLow
								THEN RobotGoVerticalPosition:=RobotGoVerticalPosition+10;
								END_IF;
								IF RobotGoVerticalPosition>=190
								THEN	RobotGoVerticalPosition:=190;
										IF NOT RobotInAssemblyUnitBlockLow
										THEN Bit3Input:=TRUE; (*1000 = RobotInAssemblyUnit*)
										END_IF;
										CaseBlack:=67;
								END_IF;
						(*Per portare il pezzo nella stazione pezzi finiti è sufficiente dare il comando di ritorno alla posizione iniziale*)
						67:		IF (NOT Bit3Output AND NOT Bit2Output AND NOT Bit1Output AND Bit0Output) AND NOT RobotGoToInitialPositionBlockLow    (*0001 = RobotGoToInitialPosition*)
								THEN CaseBlack:=68;
								ELSE CaseBlack:=67;
								END_IF;

						68 :	ElementInEndEffectorRed:=ElementAssemblyRed;
								ElementInEndEffectorBlack:=ElementAssemblyBlack;
								ElementInEndEffectorSilver:=ElementAssemblySilver;
								ElementInEndEffector:=TRUE;
								PistonBlackInEndEffector:=PistonBlackAssembly;
								PistonSilverInEndEffector:=PistonSilverAssembly;
								CaseBlack:=69;

						69:		CoverAssembly:=FALSE;
								SpringAssembly:=FALSE;
								PistonBlackAssembly:=FALSE;
								PistonSilverAssembly:=FALSE;
								ElementAssemblyBlack:=FALSE;
								ElementAssemblySilver:=FALSE;
								ElementAssemblyRed:=FALSE;
								CaseBlack:=70;

						70:		IF NOT RobotEngineBlockLow
								THEN RobotGoVerticalPosition:=RobotGoVerticalPosition-10; (*SALI IN DIREZIONE VERTICALE*)
								END_IF;
								IF NOT RobotInAssemblyUnitBlockHigh
								THEN Bit3Input:=FALSE; (*RobotInAssemblyUnit:=FALSE*)
								END_IF;
								IF RobotGoVerticalPosition<=0
								THEN 	RobotGoVerticalPosition:=0;
										CaseBlack:=71;
								END_IF;

						71: 	CanText:='Pezzi Finiti'; (*SCRITTA "Pezzi Finiti" ALL'INTERNO DEL CESTO*)
								CanColour:=TRUE; (* CESTO VERDE*)
								CanDiscard:=TRUE; (*VARIABILE DI VISUALIZZAZIONE: rende visibile il cesto contenente i pezzi finiti*)
								ElementToDiscard:=TRUE;	(*MOSTRA IL PEZZO CHE FINIRA' NELLA STAZIONE DI SCARTO*)
								ElementToDiscardO:='';
								ElementToDiscardRed:=ElementInEndEffectorRed;
								ElementToDiscardBlack:=ElementInEndEffectorBlack;
								ElementToDiscardSilver:=ElementInEndEffectorSilver;
								IF CoverInEndEffector
								THEN CoverToDiscard:=TRUE; (*MOSTRA IL COPERCHIO*)
								END_IF;
								PistonBlackToDiscard:=PistonBlackInEndEffector;
								PistonSilverToDiscard:=PistonSilverInEndEffector;
								CaseBlack:=72;

						72:		EndEffectorPosition:=EndEffectorPosition-1; (*APRI END-EFFECTOR*)
								IF EndEffectorPosition<=0
								THEN 	EndEffectorPosition:=0;
										CaseBlack:=73;
								END_IF;

						73: 	ElementInEndEffector:=FALSE; (*RENDO INVISIBILE LA BASE NELL'END-EFFECTOR*)
								ElementInEndEffectorRed:=FALSE; (*RESET DELLE BASI NELL'END-EFFECTOR, NON L'HO FATTO NELL'IF PRECEDENTE PERCHE' AVREI RESO INVISIBILI LE BASI NELLA STAZIONE SCARTI*)
								ElementInEndEffectorBlack:=FALSE;
								ElementInEndEffectorSilver:=FALSE;
								ElementInEndEffectorOverturned:=FALSE;
								CoverInEndEffector:=FALSE;
								PistonBlackInEndEffector:=FALSE;
								PistonSilverInEndEffector:=FALSE;
								CaseBlack:=74;

						74:		ElementToDiscardPosition:=ElementToDiscardPosition+4; (*lo scarto scende fino a finire nel cestino*)
								IF ElementToDiscardPosition>=80
								THEN 	ElementToDiscardPosition:=80;
										CaseBlack:=75;
								END_IF;

						75:		IF NOT RobotEngineBlockLow
								THEN RobotGoHorizontalPosition:=RobotGoHorizontalPosition-10;
								END_IF;
								IF RobotGoHorizontalPosition<=0
								THEN 	RobotGoHorizontalPosition:=0;
										CaseBlack:=76;
								END_IF;

						76:		ElementAssembled:=TRUE;
								IF NOT RobotInInitialPositionBlockLow
								THEN Bit1Input:=TRUE; Bit0Input:=TRUE; (*RobotInInitialPosition:=TRUE; *)
								END_IF;
								State:=0;
	END_CASE;




3:	CASE CaseRedSilver OF

							(*Preleva la base rossa-argento*)
						20:		IF NOT RobotEngineBlockLow
								THEN RobotGoVerticalPosition:=RobotGoVerticalPosition+10; (*SCENDI SECONDO LA DIREZIONE VERTICALE*)
								END_IF;
								IF RobotGoVerticalPosition>=170
								THEN	RobotGoVerticalPosition:=170;
										CaseRedSilver:=21;
								END_IF;

						21:		EndEffectorPosition:=EndEffectorPosition+1; (*CHIUDI END-EFFECTOR*)
								IF EndEffectorPosition>=3
								THEN 	EndEffectorPosition:=3;
										CaseRedSilver:=22;
								END_IF;

						22:		ElementInEndEffector:=TRUE; (*MOSTRA LA BASE NELL'END-EFFECTOR*)
								ElementInEndEffectorBlack:=ElementStation1RobotBlack;
								ElementInEndEffectorSilver:=ElementStation1RobotSilver;
								ElementInEndEffectorRed:=ElementStation1RobotRed;
								ElementInEndEffectorOverturned:=ElementStation1RobotOverturned;
								IF ElementInEndEffectorOverturned
								THEN ElementInEndEffectorO:='O';
								ELSE ElementInEndEffectorO:='';
								END_IF;
								CaseRedSilver:=23;

						23:		ElementStation1RobotCharged:=FALSE;
								CaseRedSilver:=24;

						24:		IF NOT RobotEngineBlockLow
								THEN RobotGoVerticalPosition:=RobotGoVerticalPosition-10; (*SALI SECONDO LA DIREZIONE VERTICALE*)
								END_IF;
								IF RobotGoVerticalPosition<=0
								THEN	RobotGoVerticalPosition:=0;
										CaseRedSilver:=25;
								END_IF;

						25:		ElementStation1RobotRed:=FALSE; (*RESETTO LE INFORMAZIONI ALLA STAZIONE1 PRIMA DI METTERE A FALSE AvailableLoadForRobot IN MODO DA AVERE LE GIUSTE INFORMAZIONI SUL PEZZO SUCCESSIVO*)
								ElementStation1RobotBlack:=FALSE;
								ElementStation1RobotSilver:=FALSE;
								ElementStation1RobotOverturned:=FALSE;
								IF NOT AvailableLoadForRobotBlockHigh
								THEN AvailableLoadForRobot:=FALSE; (*RESET DEL SENSORE DI PRESENZA NELLA STAZIONE1, A QUESTO PUNTO LA GIOSTRA PUO' MANDARE UN'ALTRO PEZZO*)
								END_IF;
								CaseRedSilver:=26;

						26 :	IF NOT RobotEngineBlockLow
								THEN RobotGoHorizontalPosition:=RobotGoHorizontalPosition+10; (*MUOVITI ORIZZONTALMENTE VERSO DESTRA*)
								END_IF;
								IF RobotGoHorizontalPosition>=100
								THEN	RobotGoHorizontalPosition:=100;
										CaseRedSilver:=27;
								END_IF;

						27 :	IF NOT RobotEngineBlockLow
								THEN RobotGoVerticalPosition:=RobotGoVerticalPosition+10; (*SCENDI SECONDO LA DIREZIONE VERTICALE*)
								END_IF;
								IF RobotGoVerticalPosition>=190
								THEN 	RobotGoVerticalPosition:=190;
										CaseRedSilver:=28;
								END_IF;

						28 :	EndEffectorPosition:=EndEffectorPosition-1; (*APRI END-EFFECTOR*)
								IF EndEffectorPosition<=0
								THEN	EndEffectorPosition:=0;
										CaseRedSilver:=29;
								END_IF;

						29:		ElementAssemblyCharged:=TRUE; (*MOSTRA LA BASE NELLA STAZIONE DI ASSEMBLAGGIO*)
								ElementAssemblyBlack:=ElementInEndEffectorBlack;
								ElementAssemblySilver:=ElementInEndEffectorSilver;
								ElementAssemblyRed:=ElementInEndEffectorRed;
								CaseRedSilver:=30;

						30 :	ElementInEndEffector:=FALSE; (*NASCONDI LA BASE SULL'END-EFFECTOR*)
								ElementInEndEffectorBlack:=FALSE;
								ElementInEndEffectorSilver:=FALSE;
								ElementInEndEffectorRed:=FALSE;
								ElementInEndEffectorOverturned:=FALSE;
								IF NOT RobotInAssemblyUnitBlockLow AND NOT RobotInInitialPositionBlockHigh
								THEN Bit3Input:=TRUE; Bit2Input:=FALSE; Bit1Input:=FALSE; Bit0Input:=FALSE; (*1000 = RobotInAssemblyUnit*)
								END_IF;
								CaseRedSilver:=31;

						31:		IF (NOT Bit3Output AND Bit2Output AND Bit1Output AND Bit0Output) AND NOT RobotGoToPistonHouseBlockLow   (*0111 = Prendi Pistone*)
								THEN CaseRedSilver:=32;
								ELSE CaseRedSilver:=31;
								END_IF;

						32 :	IF NOT RobotEngineBlockLow
								THEN RobotGoVerticalPosition:=RobotGoVerticalPosition-10;
								END_IF;
								IF NOT RobotInAssemblyUnitBlockHigh
								THEN Bit3Input:=FALSE; (*RobotInAssemblyUnit:=FALSE*)
								END_IF;
								IF RobotGoVerticalPosition<=-110
								THEN	RobotGoVerticalPosition:=-110;
										CaseRedSilver:=33;
								END_IF;

						33 :	EndEffectorPosition:=EndEffectorPosition+2; (*CHIUDI END-EFFECTOR PER POTER PASSARE TRA LE DUE TORRETTE DEI PISTONI*)
								IF EndEffectorPosition>=20
								THEN 	EndEffectorPosition:=20;
										CaseRedSilver:=34;
								END_IF;

						34 :	IF NOT RobotEngineBlockLow
								THEN RobotGoHorizontalPosition:=RobotGoHorizontalPosition+10;
								END_IF;
								IF RobotGoHorizontalPosition>=435
								THEN 	RobotGoHorizontalPosition:=435;
										CaseRedSilver:=35;
								END_IF;

						35 : 	IF NOT RobotEngineBlockLow
								THEN RobotGoVerticalPosition:=RobotGoVerticalPosition+10;
								END_IF;
								IF RobotGoVerticalPosition>=230
								THEN	RobotGoVerticalPosition:=230;
										CaseRedSilver:=36;
								END_IF;

						36 :	EndEffectorPosition:=EndEffectorPosition+2; (*CHIUDI END-EFFECTOR PER PRESA PISTONE*)
								IF EndEffectorPosition>=25
								THEN 	EndEffectorPosition:=25;
										CaseRedSilver:=37;
								END_IF;

						37:		IF PistonBlackExtract AND PistonSelectorPosition=20(*NOT PistonSelectorIsOnTheRightBlockHigh AND NOT PistonSelectorIsOnTheRightBlockLow AND NOT PistonSelectorIsOnTheLeftBlockHigh AND NOT PistonSelectorIsOnTheLeftBlockLow AND NOT PistonSelectorGoOnTheRightBlockHigh AND NOT PistonSelectorGoOnTheRightBlockLow AND NOT PistonSelectorGoOnTheLeftBlockHigh AND NOT PistonSelectorGoOnTheLeftBlockLow*)
								THEN	PistonBlackInEndEffector:=TRUE; (*RENDO VISIBILE IL PISTONE NERO NELL'END-EFFECTOR*)
										PistonBlackExtract:=FALSE; (*RENDO INVISIBILE IL PISTONE NERO NEL MAGAZZINO*)
										PistonBlackNumber:=PistonBlackNumber-1;
								END_IF;
								IF NOT RobotInPistonWarehouseBlockLow
								THEN Bit0Input:=TRUE; (*RobotInPistonWarehouse:=TRUE;*)
								END_IF;
								CaseRedSilver:=38;

						38:		IF (Bit3Output AND NOT Bit2Output AND NOT Bit1Output AND Bit0Output) AND NOT RobotTakeCurrentLoadToAssemblyBlockLow  (*1001 = TakeCurrentLoadToAssemblyStation*)
								THEN CaseRedSilver:=39;
								ELSE CaseRedSilver:=38;
								END_IF;

						39 :	IF NOT RobotEngineBlockLow
								THEN RobotGoVerticalPosition:=RobotGoVerticalPosition-10;
								END_IF;
								IF NOT RobotInPistonWarehouseBlockHigh
								THEN Bit0Input:=FALSE; (*RobotInPistonWarehouse:=FALSE;*)
								END_IF;
								IF RobotGoVerticalPosition<=-110
								THEN	RobotGoVerticalPosition:=-110;
										CaseRedSilver:=40;
								END_IF;

						40 :	IF NOT RobotEngineBlockLow
								THEN RobotGoHorizontalPosition:=RobotGoHorizontalPosition-10;
								END_IF;
								IF RobotGoHorizontalPosition<=100
								THEN 	RobotGoHorizontalPosition:=100;
										CaseRedSilver:=41;
								END_IF;

						41 :	IF NOT RobotEngineBlockLow
								THEN RobotGoVerticalPosition:=RobotGoVerticalPosition+10;
								END_IF;
								IF RobotGoVerticalPosition>=185
								THEN	RobotGoVerticalPosition:=185;
										CaseRedSilver:=42;
								END_IF;

						42 :	EndEffectorPosition:=EndEffectorPosition-2; (*APRO END-EFFECTOR*)
								IF EndEffectorPosition<=16
								THEN 	EndEffectorPosition:=16;
										PistonBlackAssembly:=PistonBlackInEndEffector;
										PistonSilverAssembly:=PistonSilverInEndEffector;
										CaseRedSilver:=43;
								END_IF;

						43 :	PistonBlackInEndEffector:=FALSE;
								PistonSilverInEndEffector:=FALSE;
								IF NOT RobotInAssemblyUnitBlockLow
								THEN Bit3Input:=TRUE;  (*RobotInAssemblyUnit:=TRUE;*)
								END_IF;
								CaseRedSilver:=44;

						44:		IF (NOT Bit3Output AND Bit2Output AND Bit1Output AND NOT Bit0Output) AND NOT RobotGoToSpringHouseBlockLow  (*0110 = RobotGoToSpringHouse*)
								THEN CaseRedSilver:=45;
								ELSE CaseRedSilver:=44;
								END_IF;

						45 :	IF NOT RobotEngineBlockLow
								THEN RobotGoVerticalPosition:=RobotGoVerticalPosition-10;
								END_IF;
								IF NOT RobotInAssemblyUnitBlockHigh
								THEN Bit3Input:=FALSE; (*RobotInAssemblyUnit:=FALSE*)
								END_IF;
								IF RobotGoVerticalPosition<=170
								THEN	RobotGoVerticalPosition:=170;
										CaseRedSilver:=46;
								END_IF;

						46 :	IF NOT RobotEngineBlockLow
								THEN RobotGoHorizontalPosition:=RobotGoHorizontalPosition+10;
								END_IF;
								IF RobotGoHorizontalPosition>=170
								THEN 	RobotGoHorizontalPosition:=170;
										CaseRedSilver:=47;
								END_IF;

						47 : 	IF NOT RobotEngineBlockLow
								THEN RobotGoVerticalPosition:=RobotGoVerticalPosition+10;
								END_IF;
								IF RobotGoVerticalPosition>=245
								THEN	RobotGoVerticalPosition:=245;
										CaseRedSilver:=48;
								END_IF;

						48 :	EndEffectorPosition:=EndEffectorPosition+2; (*CHIUDI END-EFFECTOR PER PRESA MOLLA*)
								IF EndEffectorPosition>=20
								THEN 	EndEffectorPosition:=20;
										CaseRedSilver:=49;
								END_IF;

						49:		IF NOT ToExtractSpringInAssemblyStationInExtensivePositionBlockHigh AND NOT ToExtractSpringInAssemblyStationInExtensivePositionBlockLow AND NOT ToExtractSpringInAssemblyStationBlockLow AND NOT ToExtractSpringInAssemblyStationBlockHigh
								THEN 	SpringInEndEffector:=TRUE; (*RENDO VISIBILE LA MOLLA NELL'END-EFFECTOR*)
										SpringExtract:=FALSE; (*RENDO INVISIBILE LA MOLLA NEL MAGAZZINO*)
								END_IF;
								IF NOT RobotInSpringWarehouseBlockLow
								THEN Bit1Input:=TRUE; (*RobotInSpringWarehouse:=TRUE;*)
								END_IF;
								CaseRedSilver:=50;

						50:		IF (Bit3Output AND NOT Bit2Output AND NOT Bit1Output AND Bit0Output) AND NOT RobotTakeCurrentLoadToAssemblyBlockLow  (*1001 = TakeCurrentLoadToAssemblyStation*)
								THEN CaseRedSilver:=51;
								ELSE CaseRedSilver:=50;
								END_IF;

						51 :	IF NOT RobotEngineBlockLow
								THEN RobotGoVerticalPosition:=RobotGoVerticalPosition-10;
								END_IF;
								IF NOT RobotInSpringWarehouseBlockHigh
								THEN Bit1Input:=FALSE; (*RobotInSpringWarehouse:=FALSE;*)
								END_IF;
								IF RobotGoVerticalPosition<=140
								THEN	RobotGoVerticalPosition:=140;
										CaseRedSilver:=52;
								END_IF;

						52 :	IF NOT RobotEngineBlockLow
								THEN RobotGoHorizontalPosition:=RobotGoHorizontalPosition-10;
								END_IF;
								IF RobotGoHorizontalPosition<=100
								THEN 	RobotGoHorizontalPosition:=100;
										CaseRedSilver:=53;
								END_IF;

						53 : 	IF NOT RobotEngineBlockLow
								THEN RobotGoVerticalPosition:=RobotGoVerticalPosition+10;
								END_IF;
								IF RobotGoVerticalPosition>=180
								THEN	RobotGoVerticalPosition:=180;
										CaseRedSilver:=54;
								END_IF;

						54 :	EndEffectorPosition:=EndEffectorPosition-2; (*APERTURA END-EFFECTOR*)
								IF EndEffectorPosition<=16
								THEN 	EndEffectorPosition:=16;
										CaseRedSilver:=55;
								END_IF;

						55:		IF NOT ToExtractSpringInAssemblyStationInExtensivePositionBlockHigh AND NOT ToExtractSpringInAssemblyStationInExtensivePositionBlockLow AND NOT ToExtractSpringInAssemblyStationBlockLow AND NOT ToExtractSpringInAssemblyStationBlockHigh
								THEN 	SpringInEndEffector:=FALSE; (*RENDO INVISIBILE LA MOLLA NELL'END-EFFECTOR*)
										SpringAssembly:=TRUE; (*RENDO VISIBILE LA MOLLA DENTRO LA BASE NELLA STAZIONE DI ASSEMBLAGGIO*)
								END_IF;
								IF NOT RobotInAssemblyUnitBlockLow
								THEN Bit3Input:=TRUE; (*1000 = RobotInAssemblyUnit*)
								END_IF;
								CaseRedSilver:=56;

						56:		IF (Bit3Output AND NOT Bit2Output AND NOT Bit1Output AND NOT Bit0Output) AND NOT RobotGoToCoverHouseBlockLow  (*1000 = RobotGoToCoverHouse*)
								THEN CaseRedSilver:=57;
								ELSE CaseRedSilver:=56;
								END_IF;

						57 :	IF NOT RobotEngineBlockLow
								THEN RobotGoVerticalPosition:=RobotGoVerticalPosition-10;
								END_IF;
								IF NOT RobotInAssemblyUnitBlockHigh
								THEN Bit3Input:=FALSE; (*RobotInAssemblyUnit:=FALSE;*)
								END_IF;
								IF RobotGoVerticalPosition<=-110
								THEN	RobotGoVerticalPosition:=-110;
										CaseRedSilver:=58;
								END_IF;

						58 :	EndEffectorPosition:=EndEffectorPosition-2; (*APERTURA END-EFFECTOR*)
								IF EndEffectorPosition<=0
								THEN 	EndEffectorPosition:=0;
										CaseRedSilver:=59;
								END_IF;

						59 :	IF NOT RobotEngineBlockLow
								THEN RobotGoHorizontalPosition:=RobotGoHorizontalPosition+10;
								END_IF;
								IF RobotGoHorizontalPosition>=500
								THEN 	RobotGoHorizontalPosition:=500;
										CaseRedSilver:=60;
								END_IF;

						60 : 	IF NOT RobotEngineBlockLow
								THEN RobotGoVerticalPosition:=RobotGoVerticalPosition+10;
								END_IF;
								IF RobotGoVerticalPosition>=250
								THEN	RobotGoVerticalPosition:=250;
										CaseRedSilver:=61;
								END_IF;

						61 :	EndEffectorPosition:=EndEffectorPosition+1; (*CHIUDI END-EFFECTOR PER PRESA MOLLA*)
								IF EndEffectorPosition>=3
								THEN 	EndEffectorPosition:=3;
										CaseRedSilver:=62;
								END_IF;

						62:		IF NOT ToExtractCoverInAssemblyStationForwardBlockLow AND NOT Count3
								THEN 	CoverInEndEffector:=TRUE; (*RENDO VISIBILE IL COPERCHIO NEL END-EFFECTOR*)
										CoverExtract:=FALSE; (*RENDO INVISIBILE IL COPERCHIO NEL MAGAZZINO*)
										IF ToExtractCoverInAssemblyStationForwardBlockHigh OR ToExtractCoverInAssemblyStationInExtensivePositionBlockHigh
										THEN Count3:=TRUE;
										END_IF;
								END_IF;
								IF NOT RobotInCoverWarehouseBlockLow
								THEN Bit2Input:=TRUE; (*RobotInCoverWarehouse:=TRUE;*)
								END_IF;
								CaseRedSilver:=63;

						63:		IF (Bit3Output AND NOT Bit2Output AND NOT Bit1Output AND Bit0Output) AND NOT RobotTakeCurrentLoadToAssemblyBlockLow   (*1001 = TakeCurrentLoadToAssemblyStation*)
								THEN CaseRedSilver:=64;
								ELSE CaseRedSilver:=63;
								END_IF;

						64 :	IF NOT RobotEngineBlockLow
								THEN RobotGoVerticalPosition:=RobotGoVerticalPosition-10;
								END_IF;
								IF NOT RobotInCoverWarehouseBlockHigh
								THEN Bit2Input:=FALSE; (*RobotInCoverWarehouse:=FALSE;*)
								END_IF;
								IF RobotGoVerticalPosition<=-110
								THEN	RobotGoVerticalPosition:=-110;
										CaseRedSilver:=65;
								END_IF;

						65 :	IF NOT RobotEngineBlockLow
								THEN RobotGoHorizontalPosition:=RobotGoHorizontalPosition-10;
								END_IF;
								IF RobotGoHorizontalPosition<=100
								THEN 	RobotGoHorizontalPosition:=100;
										CaseRedSilver:=66;
								END_IF;

						66 : 	IF NOT RobotEngineBlockLow
								THEN RobotGoVerticalPosition:=RobotGoVerticalPosition+10;
								END_IF;
								IF RobotGoVerticalPosition>=190
								THEN	RobotGoVerticalPosition:=190;
										IF NOT RobotInAssemblyUnitBlockLow
										THEN Bit3Input:=TRUE; (*1000 = RobotInAssemblyUnit*)
										END_IF;
										CaseRedSilver:=67;
								END_IF;
						(*Per portare il pezzo nella stazione pezzi finiti è sufficiente dare il comando di ritorno alla posizione iniziale*)
						67:		IF (NOT Bit3Output AND NOT Bit2Output AND NOT Bit1Output AND Bit0Output) AND NOT RobotGoToInitialPositionBlockLow  (*0001 = RobotGoToInitialPosition*)
								THEN CaseRedSilver:=68;
								ELSE CaseRedSilver:=67;
								END_IF;

						68 :	ElementInEndEffectorRed:=ElementAssemblyRed;
								ElementInEndEffectorBlack:=ElementAssemblyBlack;
								ElementInEndEffectorSilver:=ElementAssemblySilver;
								ElementInEndEffector:=TRUE;
								PistonBlackInEndEffector:=PistonBlackAssembly;
								PistonSilverInEndEffector:=PistonSilverAssembly;
								CaseRedSilver:=69;

						69:		CoverAssembly:=FALSE;
								SpringAssembly:=FALSE;
								PistonBlackAssembly:=FALSE;
								PistonSilverAssembly:=FALSE;
								ElementAssemblyBlack:=FALSE;
								ElementAssemblySilver:=FALSE;
								ElementAssemblyRed:=FALSE;
								CaseRedSilver:=70;

						70:		IF NOT RobotEngineBlockLow
								THEN RobotGoVerticalPosition:=RobotGoVerticalPosition-10; (*SALI IN DIREZIONE VERTICALE*)
								END_IF;
								IF NOT RobotInAssemblyUnitBlockHigh
								THEN Bit3Input:=FALSE; (*RobotInAssemblyUnit:=FALSE*)
								END_IF;
								IF RobotGoVerticalPosition<=0
								THEN 	RobotGoVerticalPosition:=0;
										CaseRedSilver:=71;
								END_IF;

						71: 	CanText:='Pezzi Finiti'; (*SCRITTA "Pezzi Finiti" ALL'INTERNO DEL CESTO*)
								CanColour:=TRUE; (* CESTO VERDE*)
								CanDiscard:=TRUE; (*VARIABILE DI VISUALIZZAZIONE: rende visibile il cesto contenente i pezzi finiti*)
								ElementToDiscard:=TRUE;	(*MOSTRA IL PEZZO CHE FINIRA' NELLA STAZIONE DI SCARTO*)
								ElementToDiscardO:='';
								ElementToDiscardRed:=ElementInEndEffectorRed;
								ElementToDiscardBlack:=ElementInEndEffectorBlack;
								ElementToDiscardSilver:=ElementInEndEffectorSilver;
								IF CoverInEndEffector
								THEN CoverToDiscard:=TRUE; (*MOSTRA IL COPERCHIO*)
								END_IF;
								PistonBlackToDiscard:=PistonBlackInEndEffector;
								PistonSilverToDiscard:=PistonSilverInEndEffector;
								CaseRedSilver:=72;

						72:		EndEffectorPosition:=EndEffectorPosition-1; (*APRI END-EFFECTOR*)
								IF EndEffectorPosition<=0
								THEN 	EndEffectorPosition:=0;
										CaseRedSilver:=73;
								END_IF;

						73: 	ElementInEndEffector:=FALSE; (*RENDO INVISIBILE LA BASE NELL'END-EFFECTOR*)
								ElementInEndEffectorRed:=FALSE; (*RESET DELLE BASI NELL'END-EFFECTOR, NON L'HO FATTO NELL'IF PRECEDENTE PERCHE' AVREI RESO INVISIBILI LE BASI NELLA STAZIONE SCARTI*)
								ElementInEndEffectorBlack:=FALSE;
								ElementInEndEffectorSilver:=FALSE;
								ElementInEndEffectorOverturned:=FALSE;
								CoverInEndEffector:=FALSE;
								PistonBlackInEndEffector:=FALSE;
								PistonSilverInEndEffector:=FALSE;
								CaseRedSilver:=74;

						74:		ElementToDiscardPosition:=ElementToDiscardPosition+4; (*lo scarto scende fino a finire nel cestino*)
								IF ElementToDiscardPosition>=80
								THEN 	ElementToDiscardPosition:=80;
										CaseRedSilver:=75;
								END_IF;

						75:		IF NOT RobotEngineBlockLow
								THEN RobotGoHorizontalPosition:=RobotGoHorizontalPosition-10;
								END_IF;
								IF RobotGoHorizontalPosition<=0
								THEN 	RobotGoHorizontalPosition:=0;
										CaseRedSilver:=76;
								END_IF;

						76:		ElementAssembled:=TRUE;
								IF NOT RobotInInitialPositionBlockLow
								THEN Bit1Input:=TRUE; Bit0Input:=TRUE; (*RobotInInitialPosition:=TRUE; *)
								END_IF;
								State:=0;

	END_CASE;

4 :	CASE InitialPosition OF

						20:		IF RobotGoVerticalPosition<0
								THEN InitialPosition:=21;
								ELSE InitialPosition:=22;
								END_IF;

						21:		IF NOT RobotEngineBlockLow
								THEN RobotGoVerticalPosition:=RobotGoVerticalPosition+10;
								END_IF;
								IF RobotGoVerticalPosition>=0
								THEN 	RobotGoVerticalPosition:=0;
										InitialPosition:=23;
								END_IF;

						22:		IF NOT RobotEngineBlockLow
								THEN RobotGoVerticalPosition:=RobotGoVerticalPosition-10;
								END_IF;
								IF RobotGoVerticalPosition<=0
								THEN 	RobotGoVerticalPosition:=0;
										InitialPosition:=23;
								END_IF;

						23:		IF NOT RobotEngineBlockLow
								THEN RobotGoHorizontalPosition:=RobotGoHorizontalPosition-10;
								END_IF;
								IF RobotGoHorizontalPosition<=0
								THEN 	RobotGoHorizontalPosition:=0;
										EndEffectorPosition:=EndEffectorPosition-1; (*CHIUDI END-EFFECTOR*)
										IF EndEffectorPosition<=0
										THEN 	EndEffectorPosition:=0;
												IF NOT RobotInInitialPositionBlockLow
												THEN Bit1Input:=TRUE; Bit0Input:=TRUE; (*RobotInInitialPosition:=TRUE; *)
												END_IF;
												State:=0;
										END_IF;

								END_IF;
	END_CASE;

END_CASE;

(*Count3 viene utilizzato nello State=62...è un contatore utilizzato per visualizzare correttemente il coperchio in magazzino in caso di bloccaggio alto del pistone*)
IF NOT ToExtractCoverInAssemblyStationForwardBlockHigh AND NOT ToExtractCoverInAssemblyStationInExtensivePositionBlockHigh
THEN 	Count3:=FALSE;
END_IF;


(*CILINDRO DI BLOCCAGGIO(Normalmente Aperto) PEZZO NELLA STAZIONE DI ASSEMBLAGGIO*)
IF FLAGBlockingCylinderForwardInAssemblyStationBlockHigh OR (BlockingCylinderForwardInAssemblyStation AND NOT BlockingCylinderForwardInAssemblyStationBlockLow)
THEN 	CylinderPositionInAssemblyUnit:=CylinderPositionInAssemblyUnit-1;
		IF BlockingCylinderForwardInAssemblyStationBlockHigh
		THEN FLAGBlockingCylinderForwardInAssemblyStationBlockHigh:=TRUE;
		ELSE FLAGBlockingCylinderForwardInAssemblyStationBlockHigh:=FALSE;
		END_IF;
ELSE CylinderPositionInAssemblyUnit:=CylinderPositionInAssemblyUnit+1;
END_IF;

IF CylinderPositionInAssemblyUnit>=6
THEN CylinderPositionInAssemblyUnit:=6;
END_IF;

IF CylinderPositionInAssemblyUnit<=0
THEN CylinderPositionInAssemblyUnit:=0;
END_IF;

IF Remove
THEN 	ElementAssembled:=TRUE;
		ElementInEndEffector:=FALSE;
		CoverInEndEffector:=FALSE;
		PistonBlackInEndEffector:=FALSE;
		PistonSilverInEndEffector:=FALSE;
		SpringInEndEffector:=FALSE;
		ElementAssemblyBlack:=FALSE;
		ElementAssemblyRed:=FALSE;
		ElementAssemblySilver:=FALSE;
		CoverAssembly:=FALSE;
		PistonBlackAssembly:=FALSE;
		PistonSilverAssembly:=FALSE;
		SpringAssembly:=FALSE;
		SpringExtract:=FALSE;
		CoverExtract:=FALSE;
		ElementStation1RobotCharged:=FALSE;
		(*FillAllWarehouses:=TRUE;*)
		AvailableLoadForRobot:=FALSE;
		IF PistonSelectorIsOnTheLeft
		THEN PistonBlackExtract:=FALSE;
		END_IF;
END_IF;
END_PROGRAM

(* POU Bridge/InputBridge, ST *)
PROGRAM InputBridge
VAR
END_VAR
(*Sensors of the 1° station*)

S_EmptyWarehouse1 :=  FaultSim(FaultLow:= EmptyWarehouseBlockedLow , FaultHigh := EmptyWarehouseBlockedHigh , Input := EmptyWarehouse);
S_CylinderExtended1 :=  FaultSim(FaultLow:= CylinderExtractionLoadInExtensivePositionBlockedLow , FaultHigh := CylinderExtractionLoadInExtensivePositionBlockedHigh , Input := CylinderExtractionLoadInExtensivePosition);
S_CylinderRetracted1 :=  FaultSim(FaultLow:= CylinderExtractionLoadInRetroactivePositionBlockedLow , FaultHigh := CylinderExtractionLoadInRetroactivePositionBlockedHigh , Input := CylinderExtractionLoadInRetroactivePosition);
S_ArmInWarehouse1 :=  FaultSim(FaultLow:= RotaryMakerInPositionWarehouseBlockedLow , FaultHigh := RotaryMakerInPositionWarehouseBlockedHigh , Input := RotaryMakerInPositionWarehouse);
S_ArmInElevator1 :=  FaultSim(FaultLow:= RotaryMakerInPositionVerificationBlockedLow , FaultHigh := RotaryMakerInPositionVerificationBlockedHigh , Input := RotaryMakerInPositionVerification);
S_VacuumOk1 :=  FaultSim(FaultLow:= VacuumGeneratorOkBlockedLow , FaultHigh := VacuumGeneratorOkBlockedHigh , Input := VacuumGeneratorOk);

(*Sensors of the 2° station*)

